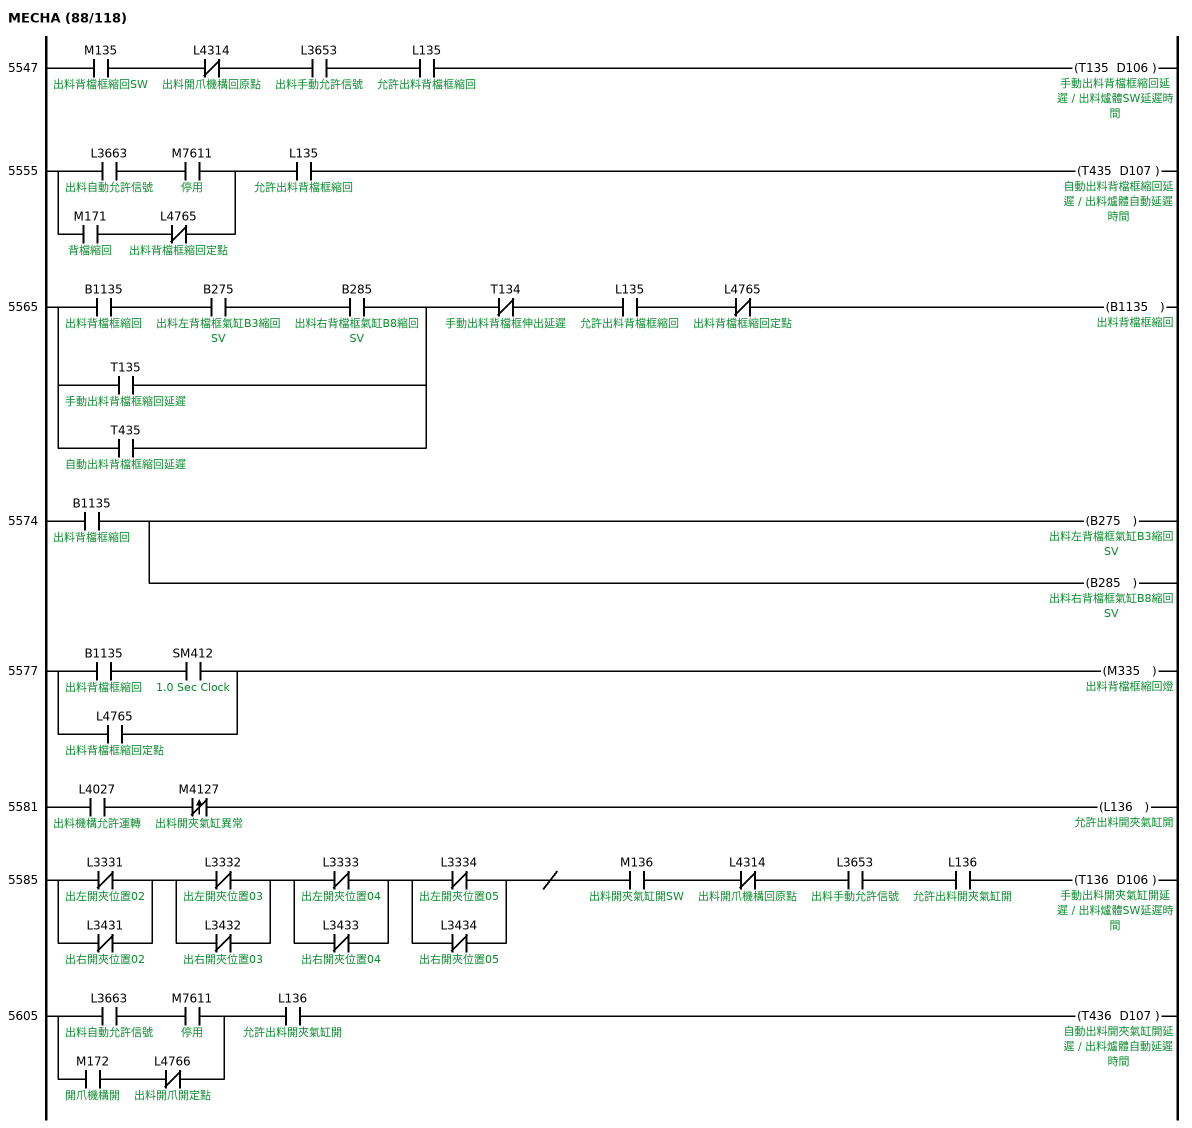
[picture p384: ladder of MECHA, rungs at steps 5547 to 5605]
5547  LD      M135  ; 出料背檔框縮回SW
      ANI     L4314  ; 出料開爪機構回原點
      AND     L3653  ; 出料手動允許信號
      AND     L135  ; 允許出料背檔框縮回
      OUT     T135 D106  ; 手動出料背檔框縮回延遲 / 出料爐體SW延遲時間
5555  LD      L3663  ; 出料自動允許信號
      AND     M7611  ; 停用
      LD      M171  ; 背檔縮回
      ANI     L4765  ; 出料背檔框縮回定點
      ORB
      AND     L135  ; 允許出料背檔框縮回
      OUT     T435 D107  ; 自動出料背檔框縮回延遲 / 出料爐體自動延遲時間
5565  LD      B1135  ; 出料背檔框縮回
      AND     B275  ; 出料左背檔框氣缸B3縮回SV
      AND     B285  ; 出料右背檔框氣缸B8縮回SV
      OR      T135  ; 手動出料背檔框縮回延遲
      OR      T435  ; 自動出料背檔框縮回延遲
      ANI     T134  ; 手動出料背檔框伸出延遲
      AND     L135  ; 允許出料背檔框縮回
      ANI     L4765  ; 出料背檔框縮回定點
      OUT     B1135  ; 出料背檔框縮回
5574  LD      B1135  ; 出料背檔框縮回
      OUT     B275  ; 出料左背檔框氣缸B3縮回SV
      OUT     B285  ; 出料右背檔框氣缸B8縮回SV
5577  LD      B1135  ; 出料背檔框縮回
      AND     SM412  ; 1.0 Sec Clock
      OR      L4765  ; 出料背檔框縮回定點
      OUT     M335  ; 出料背檔框縮回燈
5581  LD      L4027  ; 出料機構允許運轉
      ANDPI   M4127  ; 出料開夾氣缸異常
      OUT     L136  ; 允許出料開夾氣缸開
5585  LDI     L3331  ; 出左開夾位置02
      ORI     L3431  ; 出右開夾位置02
      LDI     L3332  ; 出左開夾位置03
      ORI     L3432  ; 出右開夾位置03
      ANB
      LDI     L3333  ; 出左開夾位置04
      ORI     L3433  ; 出右開夾位置04
      ANB
      LDI     L3334  ; 出左開夾位置05
      ORI     L3434  ; 出右開夾位置05
      ANB
      INV
      AND     M136  ; 出料開夾氣缸開SW
      ANI     L4314  ; 出料開爪機構回原點
      AND     L3653  ; 出料手動允許信號
      AND     L136  ; 允許出料開夾氣缸開
      OUT     T136 D106  ; 手動出料開夾氣缸開延遲 / 出料爐體SW延遲時間
5605  LD      L3663  ; 出料自動允許信號
      AND     M7611  ; 停用
      LD      M172  ; 開爪機構開
      ANI     L4766  ; 出料開爪開定點
      ORB
      AND     L136  ; 允許出料開夾氣缸開
      OUT     T436 D107  ; 自動出料開夾氣缸開延遲 / 出料爐體自動延遲時間
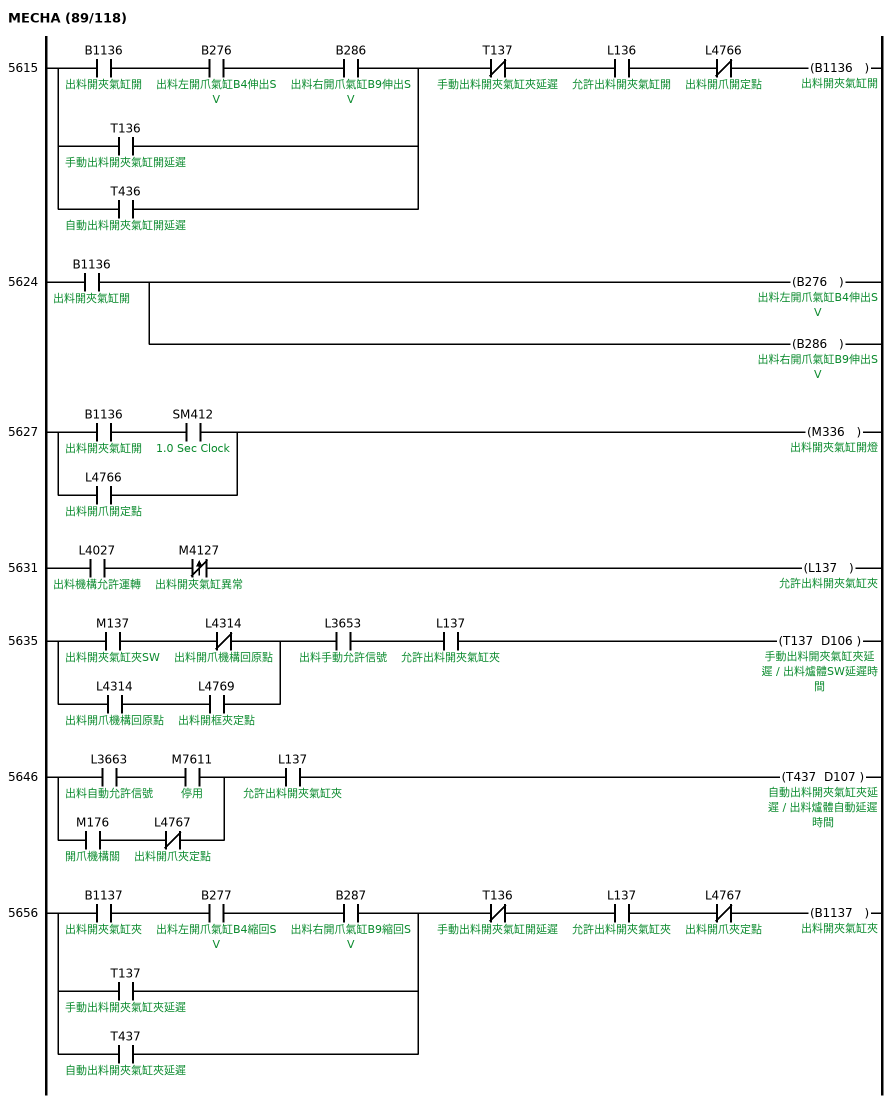
5615  LD      B1136  ; 出料開夾氣缸開
      AND     B276  ; 出料左開爪氣缸B4伸出SV
      AND     B286  ; 出料右開爪氣缸B9伸出SV
      OR      T136  ; 手動出料開夾氣缸開延遲
      OR      T436  ; 自動出料開夾氣缸開延遲
      ANI     T137  ; 手動出料開夾氣缸夾延遲
      AND     L136  ; 允許出料開夾氣缸開
      ANI     L4766  ; 出料開爪開定點
      OUT     B1136  ; 出料開夾氣缸開
5624  LD      B1136  ; 出料開夾氣缸開
      OUT     B276  ; 出料左開爪氣缸B4伸出SV
      OUT     B286  ; 出料右開爪氣缸B9伸出SV
5627  LD      B1136  ; 出料開夾氣缸開
      AND     SM412  ; 1.0 Sec Clock
      OR      L4766  ; 出料開爪開定點
      OUT     M336  ; 出料開夾氣缸開燈
5631  LD      L4027  ; 出料機構允許運轉
      ANDPI   M4127  ; 出料開夾氣缸異常
      OUT     L137  ; 允許出料開夾氣缸夾
5635  LD      M137  ; 出料開夾氣缸夾SW
      ANI     L4314  ; 出料開爪機構回原點
      LD      L4314  ; 出料開爪機構回原點
      AND     L4769  ; 出料開框夾定點
      ORB
      AND     L3653  ; 出料手動允許信號
      AND     L137  ; 允許出料開夾氣缸夾
      OUT     T137 D106  ; 手動出料開夾氣缸夾延遲 / 出料爐體SW延遲時間
5646  LD      L3663  ; 出料自動允許信號
      AND     M7611  ; 停用
      LD      M176  ; 開爪機構關
      ANI     L4767  ; 出料開爪夾定點
      ORB
      AND     L137  ; 允許出料開夾氣缸夾
      OUT     T437 D107  ; 自動出料開夾氣缸夾延遲 / 出料爐體自動延遲時間
5656  LD      B1137  ; 出料開夾氣缸夾
      AND     B277  ; 出料左開爪氣缸B4縮回SV
      AND     B287  ; 出料右開爪氣缸B9縮回SV
      OR      T137  ; 手動出料開夾氣缸夾延遲
      OR      T437  ; 自動出料開夾氣缸夾延遲
      ANI     T136  ; 手動出料開夾氣缸開延遲
      AND     L137  ; 允許出料開夾氣缸夾
      ANI     L4767  ; 出料開爪夾定點
      OUT     B1137  ; 出料開夾氣缸夾
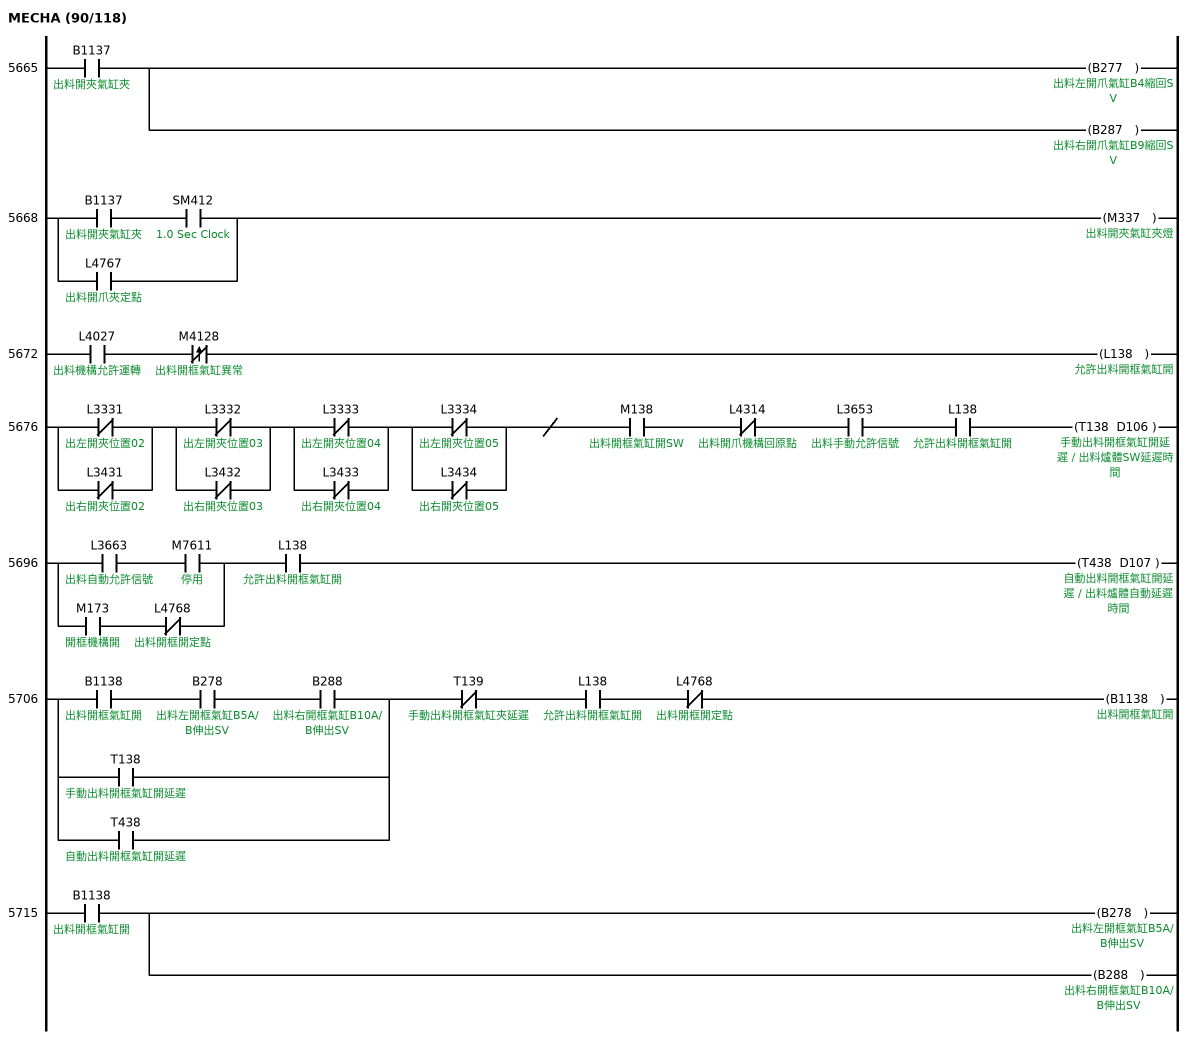
5665  LD      B1137  ; 出料開夾氣缸夾
      OUT     B277  ; 出料左開爪氣缸B4縮回SV
      OUT     B287  ; 出料右開爪氣缸B9縮回SV
5668  LD      B1137  ; 出料開夾氣缸夾
      AND     SM412  ; 1.0 Sec Clock
      OR      L4767  ; 出料開爪夾定點
      OUT     M337  ; 出料開夾氣缸夾燈
5672  LD      L4027  ; 出料機構允許運轉
      ANDPI   M4128  ; 出料開框氣缸異常
      OUT     L138  ; 允許出料開框氣缸開
5676  LDI     L3331  ; 出左開夾位置02
      ORI     L3431  ; 出右開夾位置02
      LDI     L3332  ; 出左開夾位置03
      ORI     L3432  ; 出右開夾位置03
      ANB
      LDI     L3333  ; 出左開夾位置04
      ORI     L3433  ; 出右開夾位置04
      ANB
      LDI     L3334  ; 出左開夾位置05
      ORI     L3434  ; 出右開夾位置05
      ANB
      INV
      AND     M138  ; 出料開框氣缸開SW
      ANI     L4314  ; 出料開爪機構回原點
      AND     L3653  ; 出料手動允許信號
      AND     L138  ; 允許出料開框氣缸開
      OUT     T138 D106  ; 手動出料開框氣缸開延遲 / 出料爐體SW延遲時間
5696  LD      L3663  ; 出料自動允許信號
      AND     M7611  ; 停用
      LD      M173  ; 開框機構開
      ANI     L4768  ; 出料開框開定點
      ORB
      AND     L138  ; 允許出料開框氣缸開
      OUT     T438 D107  ; 自動出料開框氣缸開延遲 / 出料爐體自動延遲時間
5706  LD      B1138  ; 出料開框氣缸開
      AND     B278  ; 出料左開框氣缸B5A/B伸出SV
      AND     B288  ; 出料右開框氣缸B10A/B伸出SV
      OR      T138  ; 手動出料開框氣缸開延遲
      OR      T438  ; 自動出料開框氣缸開延遲
      ANI     T139  ; 手動出料開框氣缸夾延遲
      AND     L138  ; 允許出料開框氣缸開
      ANI     L4768  ; 出料開框開定點
      OUT     B1138  ; 出料開框氣缸開
5715  LD      B1138  ; 出料開框氣缸開
      OUT     B278  ; 出料左開框氣缸B5A/B伸出SV
      OUT     B288  ; 出料右開框氣缸B10A/B伸出SV
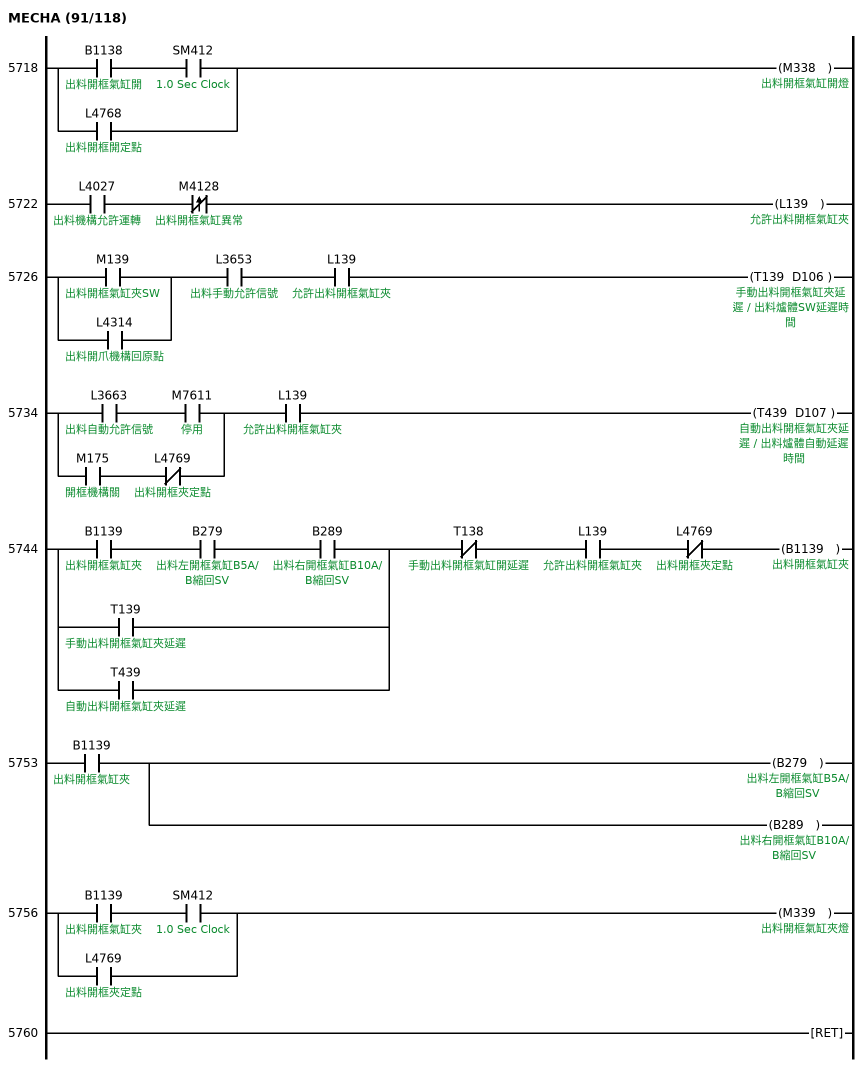
5718  LD      B1138  ; 出料開框氣缸開
      AND     SM412  ; 1.0 Sec Clock
      OR      L4768  ; 出料開框開定點
      OUT     M338  ; 出料開框氣缸開燈
5722  LD      L4027  ; 出料機構允許運轉
      ANDPI   M4128  ; 出料開框氣缸異常
      OUT     L139  ; 允許出料開框氣缸夾
5726  LD      M139  ; 出料開框氣缸夾SW
      OR      L4314  ; 出料開爪機構回原點
      AND     L3653  ; 出料手動允許信號
      AND     L139  ; 允許出料開框氣缸夾
      OUT     T139 D106  ; 手動出料開框氣缸夾延遲 / 出料爐體SW延遲時間
5734  LD      L3663  ; 出料自動允許信號
      AND     M7611  ; 停用
      LD      M175  ; 開框機構關
      ANI     L4769  ; 出料開框夾定點
      ORB
      AND     L139  ; 允許出料開框氣缸夾
      OUT     T439 D107  ; 自動出料開框氣缸夾延遲 / 出料爐體自動延遲時間
5744  LD      B1139  ; 出料開框氣缸夾
      AND     B279  ; 出料左開框氣缸B5A/B縮回SV
      AND     B289  ; 出料右開框氣缸B10A/B縮回SV
      OR      T139  ; 手動出料開框氣缸夾延遲
      OR      T439  ; 自動出料開框氣缸夾延遲
      ANI     T138  ; 手動出料開框氣缸開延遲
      AND     L139  ; 允許出料開框氣缸夾
      ANI     L4769  ; 出料開框夾定點
      OUT     B1139  ; 出料開框氣缸夾
5753  LD      B1139  ; 出料開框氣缸夾
      OUT     B279  ; 出料左開框氣缸B5A/B縮回SV
      OUT     B289  ; 出料右開框氣缸B10A/B縮回SV
5756  LD      B1139  ; 出料開框氣缸夾
      AND     SM412  ; 1.0 Sec Clock
      OR      L4769  ; 出料開框夾定點
      OUT     M339  ; 出料開框氣缸夾燈
5760  RET
      P1061
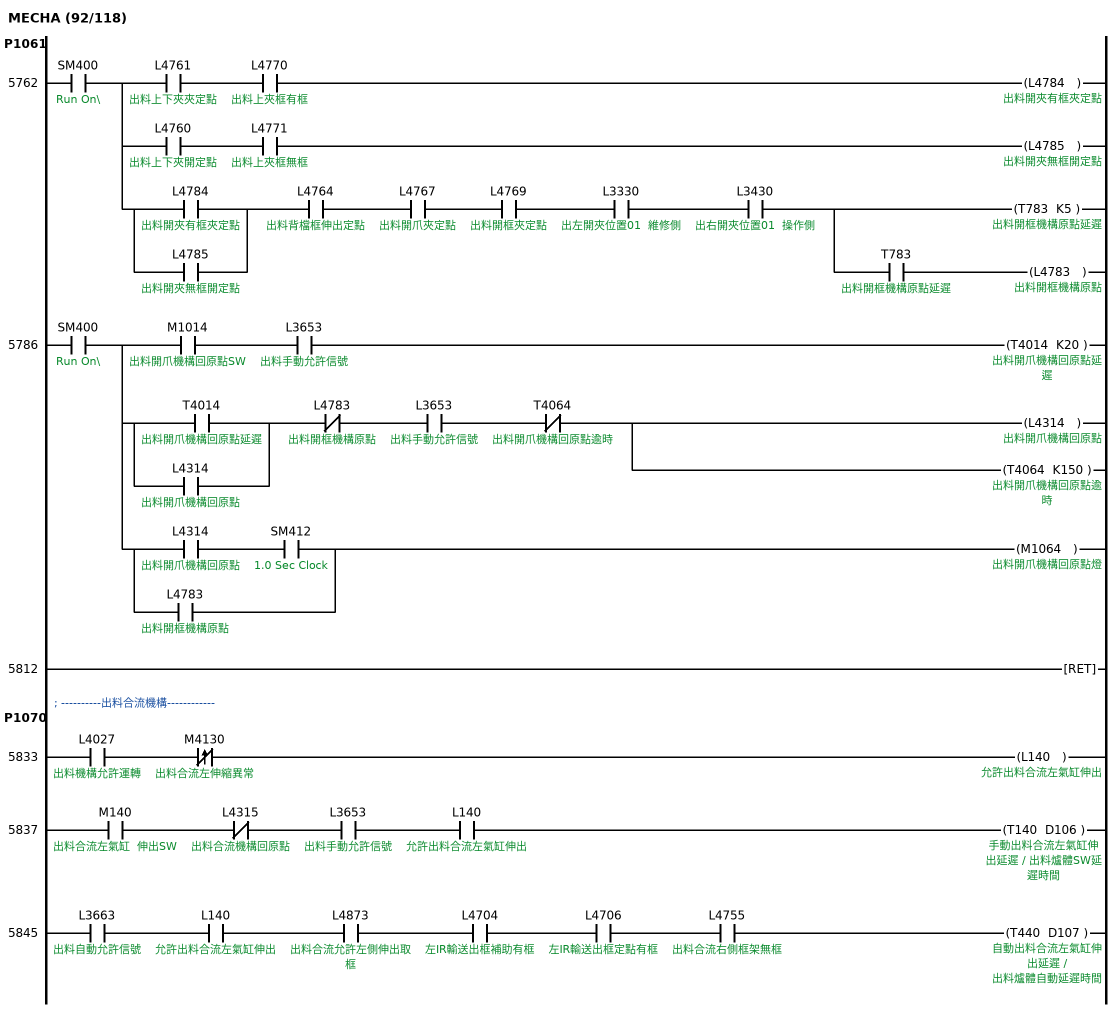
5762  LD      SM400  ; Run On\
      MPS
      AND     L4761  ; 出料上下夾夾定點
      AND     L4770  ; 出料上夾框有框
      OUT     L4784  ; 出料開夾有框夾定點
      MRD
      AND     L4760  ; 出料上下夾開定點
      AND     L4771  ; 出料上夾框無框
      OUT     L4785  ; 出料開夾無框開定點
      MPP
      LD      L4784  ; 出料開夾有框夾定點
      OR      L4785  ; 出料開夾無框開定點
      ANB
      AND     L4764  ; 出料背檔框伸出定點
      AND     L4767  ; 出料開爪夾定點
      AND     L4769  ; 出料開框夾定點
      AND     L3330  ; 出左開夾位置01  維修側
      AND     L3430  ; 出右開夾位置01  操作側
      OUT     T783 K5  ; 出料開框機構原點延遲
      AND     T783  ; 出料開框機構原點延遲
      OUT     L4783  ; 出料開框機構原點
5786  LD      SM400  ; Run On\
      MPS
      AND     M1014  ; 出料開爪機構回原點SW
      AND     L3653  ; 出料手動允許信號
      OUT     T4014 K20  ; 出料開爪機構回原點延遲
      MRD
      LD      T4014  ; 出料開爪機構回原點延遲
      OR      L4314  ; 出料開爪機構回原點
      ANB
      ANI     L4783  ; 出料開框機構原點
      AND     L3653  ; 出料手動允許信號
      ANI     T4064  ; 出料開爪機構回原點逾時
      OUT     L4314  ; 出料開爪機構回原點
      OUT     T4064 K150  ; 出料開爪機構回原點逾時
      MPP
      LD      L4314  ; 出料開爪機構回原點
      AND     SM412  ; 1.0 Sec Clock
      OR      L4783  ; 出料開框機構原點
      ANB
      OUT     M1064  ; 出料開爪機構回原點燈
5812  RET
; ----------出料合流機構------------
      P1070
5833  LD      L4027  ; 出料機構允許運轉
      ANDPI   M4130  ; 出料合流左伸縮異常
      OUT     L140  ; 允許出料合流左氣缸伸出
5837  LD      M140  ; 出料合流左氣缸  伸出SW
      ANI     L4315  ; 出料合流機構回原點
      AND     L3653  ; 出料手動允許信號
      AND     L140  ; 允許出料合流左氣缸伸出
      OUT     T140 D106  ; 手動出料合流左氣缸伸出延遲 / 出料爐體SW延遲時間
5845  LD      L3663  ; 出料自動允許信號
      AND     L140  ; 允許出料合流左氣缸伸出
      AND     L4873  ; 出料合流允許左側伸出取框
      AND     L4704  ; 左IR輸送出框補助有框
      AND     L4706  ; 左IR輸送出框定點有框
      AND     L4755  ; 出料合流右側框架無框
      OUT     T440 D107  ; 自動出料合流左氣缸伸出延遲 / 出料爐體自動延遲時間
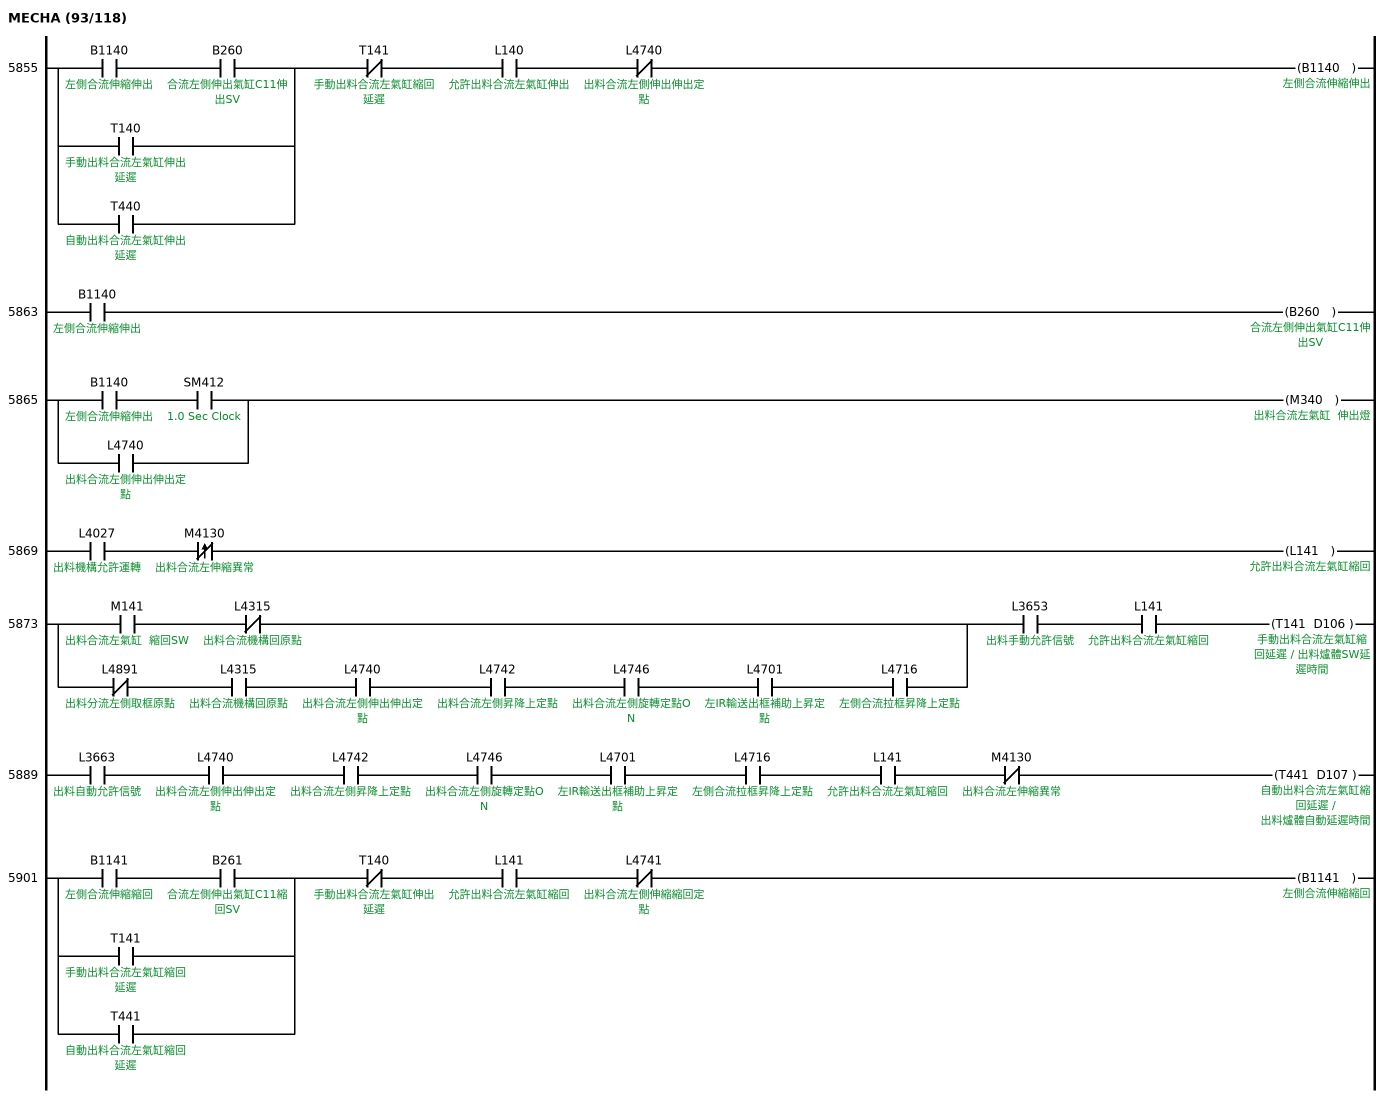
5855  LD      B1140  ; 左側合流伸縮伸出
      AND     B260  ; 合流左側伸出氣缸C11伸出SV
      OR      T140  ; 手動出料合流左氣缸伸出延遲
      OR      T440  ; 自動出料合流左氣缸伸出延遲
      ANI     T141  ; 手動出料合流左氣缸縮回延遲
      AND     L140  ; 允許出料合流左氣缸伸出
      ANI     L4740  ; 出料合流左側伸出伸出定點
      OUT     B1140  ; 左側合流伸縮伸出
5863  LD      B1140  ; 左側合流伸縮伸出
      OUT     B260  ; 合流左側伸出氣缸C11伸出SV
5865  LD      B1140  ; 左側合流伸縮伸出
      AND     SM412  ; 1.0 Sec Clock
      OR      L4740  ; 出料合流左側伸出伸出定點
      OUT     M340  ; 出料合流左氣缸  伸出燈
5869  LD      L4027  ; 出料機構允許運轉
      ANDPI   M4130  ; 出料合流左伸縮異常
      OUT     L141  ; 允許出料合流左氣缸縮回
5873  LD      M141  ; 出料合流左氣缸  縮回SW
      ANI     L4315  ; 出料合流機構回原點
      LDI     L4891  ; 出料分流左側取框原點
      AND     L4315  ; 出料合流機構回原點
      AND     L4740  ; 出料合流左側伸出伸出定點
      AND     L4742  ; 出料合流左側昇降上定點
      AND     L4746  ; 出料合流左側旋轉定點ON
      AND     L4701  ; 左IR輸送出框補助上昇定點
      AND     L4716  ; 左側合流拉框昇降上定點
      ORB
      AND     L3653  ; 出料手動允許信號
      AND     L141  ; 允許出料合流左氣缸縮回
      OUT     T141 D106  ; 手動出料合流左氣缸縮回延遲 / 出料爐體SW延遲時間
5889  LD      L3663  ; 出料自動允許信號
      AND     L4740  ; 出料合流左側伸出伸出定點
      AND     L4742  ; 出料合流左側昇降上定點
      AND     L4746  ; 出料合流左側旋轉定點ON
      AND     L4701  ; 左IR輸送出框補助上昇定點
      AND     L4716  ; 左側合流拉框昇降上定點
      AND     L141  ; 允許出料合流左氣缸縮回
      ANI     M4130  ; 出料合流左伸縮異常
      OUT     T441 D107  ; 自動出料合流左氣缸縮回延遲 / 出料爐體自動延遲時間
5901  LD      B1141  ; 左側合流伸縮縮回
      AND     B261  ; 合流左側伸出氣缸C11縮回SV
      OR      T141  ; 手動出料合流左氣缸縮回延遲
      OR      T441  ; 自動出料合流左氣缸縮回延遲
      ANI     T140  ; 手動出料合流左氣缸伸出延遲
      AND     L141  ; 允許出料合流左氣缸縮回
      ANI     L4741  ; 出料合流左側伸縮縮回定點
      OUT     B1141  ; 左側合流伸縮縮回
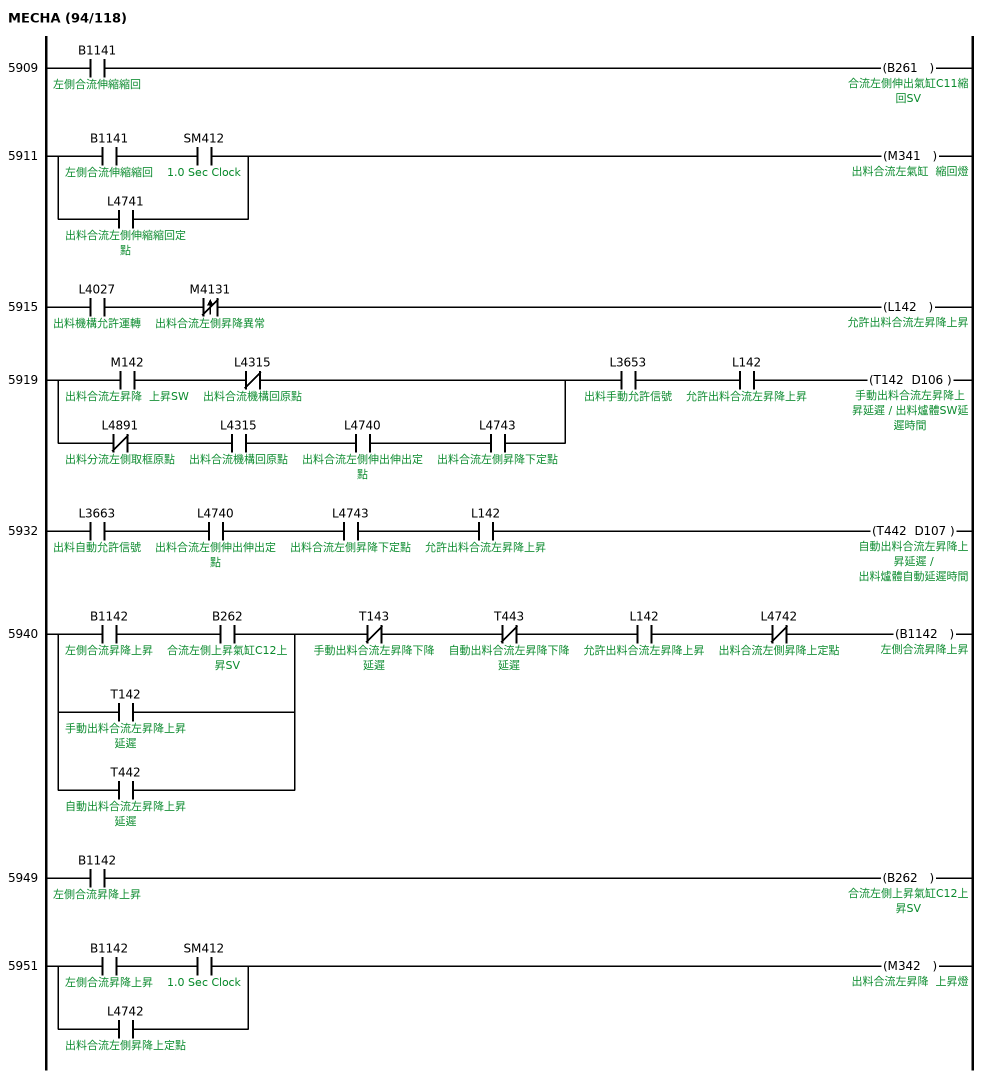
5909  LD      B1141  ; 左側合流伸縮縮回
      OUT     B261  ; 合流左側伸出氣缸C11縮回SV
5911  LD      B1141  ; 左側合流伸縮縮回
      AND     SM412  ; 1.0 Sec Clock
      OR      L4741  ; 出料合流左側伸縮縮回定點
      OUT     M341  ; 出料合流左氣缸  縮回燈
5915  LD      L4027  ; 出料機構允許運轉
      ANDPI   M4131  ; 出料合流左側昇降異常
      OUT     L142  ; 允許出料合流左昇降上昇
5919  LD      M142  ; 出料合流左昇降  上昇SW
      ANI     L4315  ; 出料合流機構回原點
      LDI     L4891  ; 出料分流左側取框原點
      AND     L4315  ; 出料合流機構回原點
      AND     L4740  ; 出料合流左側伸出伸出定點
      AND     L4743  ; 出料合流左側昇降下定點
      ORB
      AND     L3653  ; 出料手動允許信號
      AND     L142  ; 允許出料合流左昇降上昇
      OUT     T142 D106  ; 手動出料合流左昇降上昇延遲 / 出料爐體SW延遲時間
5932  LD      L3663  ; 出料自動允許信號
      AND     L4740  ; 出料合流左側伸出伸出定點
      AND     L4743  ; 出料合流左側昇降下定點
      AND     L142  ; 允許出料合流左昇降上昇
      OUT     T442 D107  ; 自動出料合流左昇降上昇延遲 / 出料爐體自動延遲時間
5940  LD      B1142  ; 左側合流昇降上昇
      AND     B262  ; 合流左側上昇氣缸C12上昇SV
      OR      T142  ; 手動出料合流左昇降上昇延遲
      OR      T442  ; 自動出料合流左昇降上昇延遲
      ANI     T143  ; 手動出料合流左昇降下降延遲
      ANI     T443  ; 自動出料合流左昇降下降延遲
      AND     L142  ; 允許出料合流左昇降上昇
      ANI     L4742  ; 出料合流左側昇降上定點
      OUT     B1142  ; 左側合流昇降上昇
5949  LD      B1142  ; 左側合流昇降上昇
      OUT     B262  ; 合流左側上昇氣缸C12上昇SV
5951  LD      B1142  ; 左側合流昇降上昇
      AND     SM412  ; 1.0 Sec Clock
      OR      L4742  ; 出料合流左側昇降上定點
      OUT     M342  ; 出料合流左昇降  上昇燈
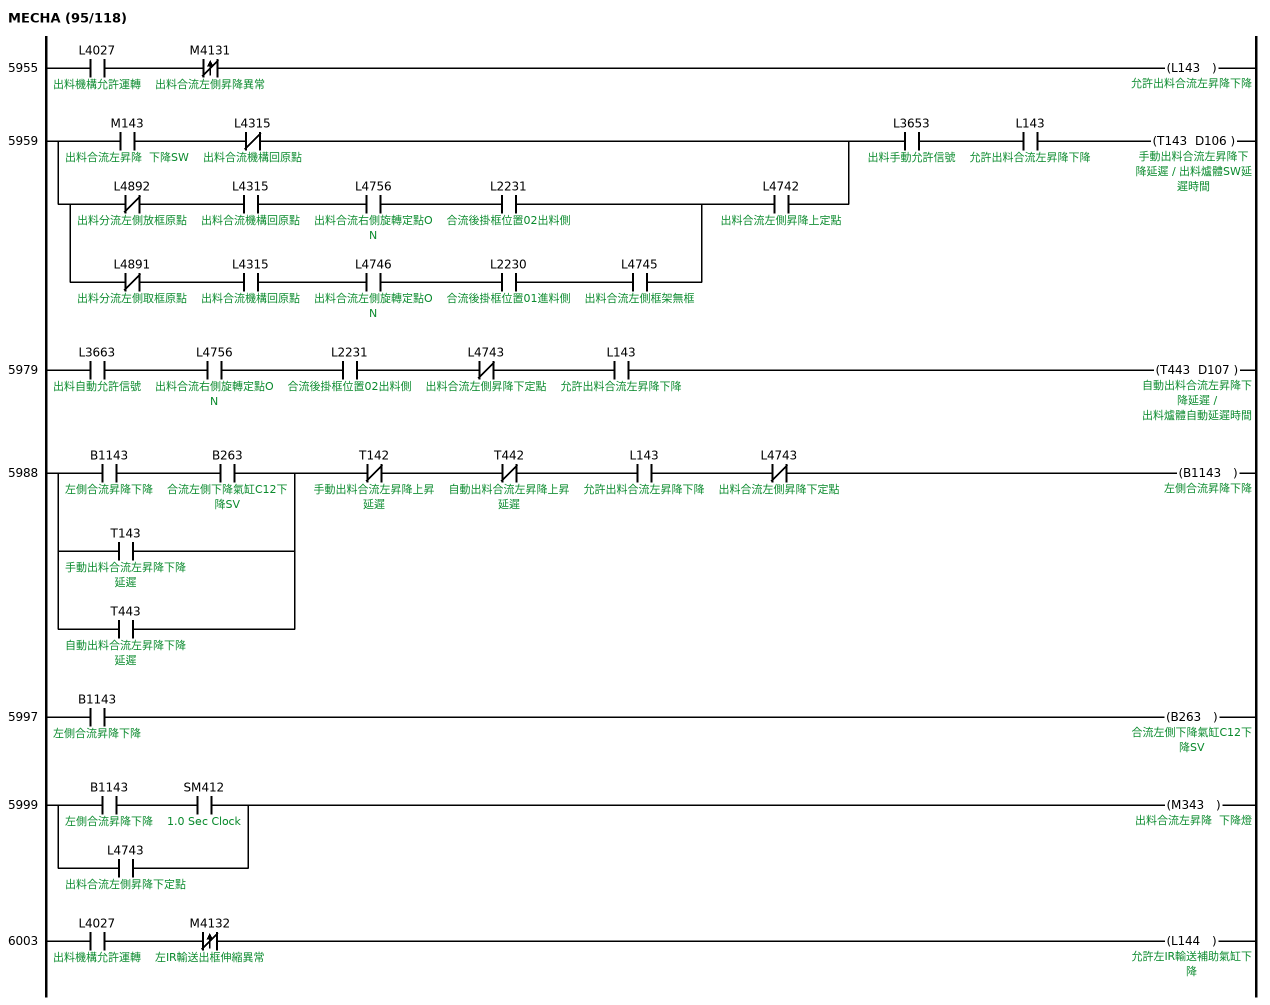
5955  LD      L4027  ; 出料機構允許運轉
      ANDPI   M4131  ; 出料合流左側昇降異常
      OUT     L143  ; 允許出料合流左昇降下降
5959  LD      M143  ; 出料合流左昇降  下降SW
      ANI     L4315  ; 出料合流機構回原點
      LDI     L4892  ; 出料分流左側放框原點
      AND     L4315  ; 出料合流機構回原點
      AND     L4756  ; 出料合流右側旋轉定點ON
      AND     L2231  ; 合流後掛框位置02出料側
      LDI     L4891  ; 出料分流左側取框原點
      AND     L4315  ; 出料合流機構回原點
      AND     L4746  ; 出料合流左側旋轉定點ON
      AND     L2230  ; 合流後掛框位置01進料側
      AND     L4745  ; 出料合流左側框架無框
      ORB
      AND     L4742  ; 出料合流左側昇降上定點
      ORB
      AND     L3653  ; 出料手動允許信號
      AND     L143  ; 允許出料合流左昇降下降
      OUT     T143 D106  ; 手動出料合流左昇降下降延遲 / 出料爐體SW延遲時間
5979  LD      L3663  ; 出料自動允許信號
      AND     L4756  ; 出料合流右側旋轉定點ON
      AND     L2231  ; 合流後掛框位置02出料側
      ANI     L4743  ; 出料合流左側昇降下定點
      AND     L143  ; 允許出料合流左昇降下降
      OUT     T443 D107  ; 自動出料合流左昇降下降延遲 / 出料爐體自動延遲時間
5988  LD      B1143  ; 左側合流昇降下降
      AND     B263  ; 合流左側下降氣缸C12下降SV
      OR      T143  ; 手動出料合流左昇降下降延遲
      OR      T443  ; 自動出料合流左昇降下降延遲
      ANI     T142  ; 手動出料合流左昇降上昇延遲
      ANI     T442  ; 自動出料合流左昇降上昇延遲
      AND     L143  ; 允許出料合流左昇降下降
      ANI     L4743  ; 出料合流左側昇降下定點
      OUT     B1143  ; 左側合流昇降下降
5997  LD      B1143  ; 左側合流昇降下降
      OUT     B263  ; 合流左側下降氣缸C12下降SV
5999  LD      B1143  ; 左側合流昇降下降
      AND     SM412  ; 1.0 Sec Clock
      OR      L4743  ; 出料合流左側昇降下定點
      OUT     M343  ; 出料合流左昇降  下降燈
6003  LD      L4027  ; 出料機構允許運轉
      ANDPI   M4132  ; 左IR輸送出框伸縮異常
      OUT     L144  ; 允許左IR輸送補助氣缸下降
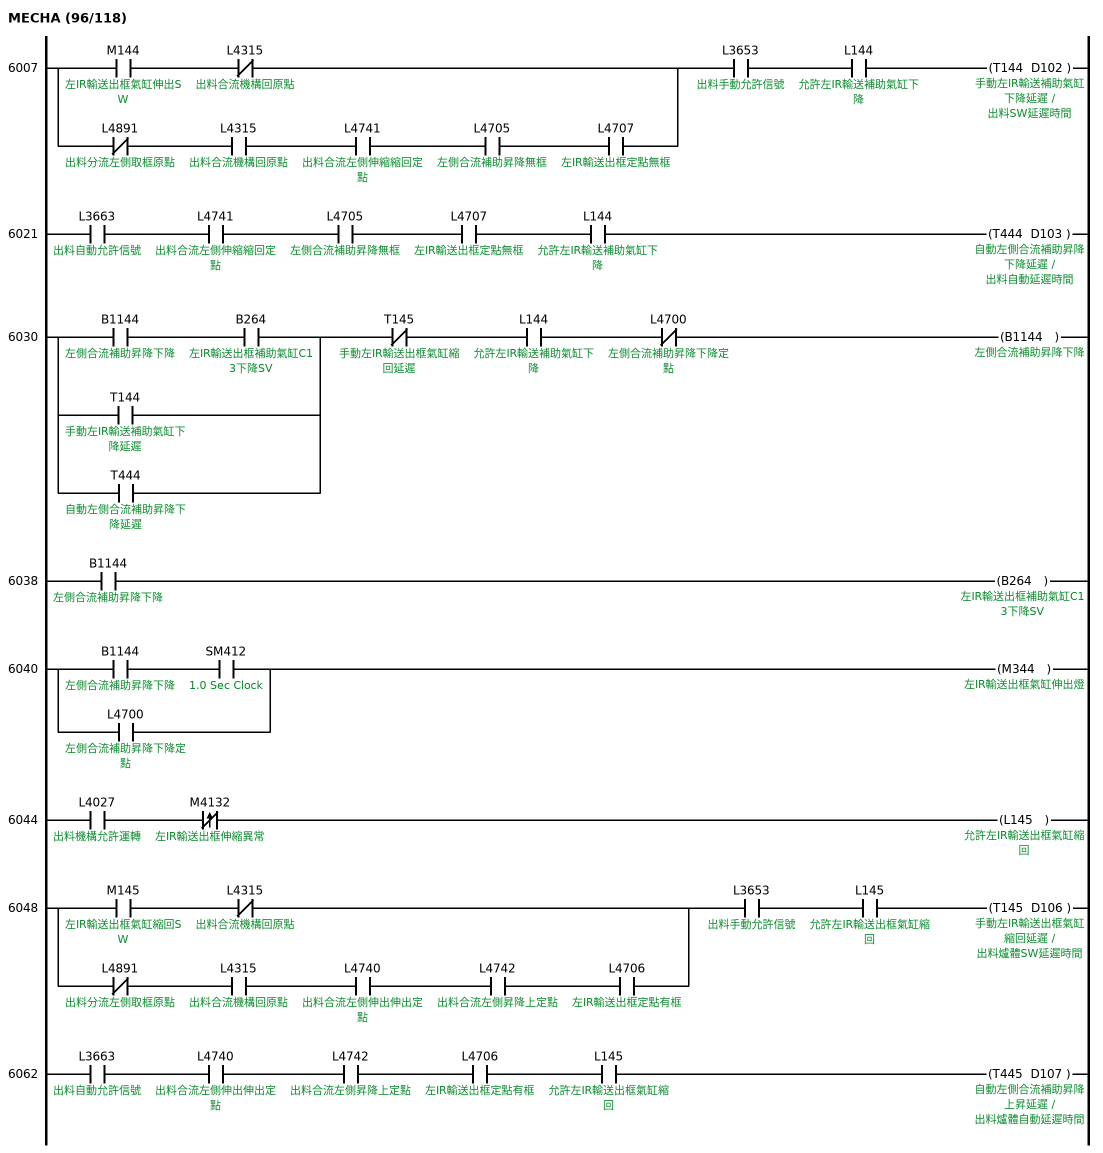
6007  LD      M144  ; 左IR輸送出框氣缸伸出SW
      ANI     L4315  ; 出料合流機構回原點
      LDI     L4891  ; 出料分流左側取框原點
      AND     L4315  ; 出料合流機構回原點
      AND     L4741  ; 出料合流左側伸縮縮回定點
      AND     L4705  ; 左側合流補助昇降無框
      AND     L4707  ; 左IR輸送出框定點無框
      ORB
      AND     L3653  ; 出料手動允許信號
      AND     L144  ; 允許左IR輸送補助氣缸下降
      OUT     T144 D102  ; 手動左IR輸送補助氣缸下降延遲 / 出料SW延遲時間
6021  LD      L3663  ; 出料自動允許信號
      AND     L4741  ; 出料合流左側伸縮縮回定點
      AND     L4705  ; 左側合流補助昇降無框
      AND     L4707  ; 左IR輸送出框定點無框
      AND     L144  ; 允許左IR輸送補助氣缸下降
      OUT     T444 D103  ; 自動左側合流補助昇降下降延遲 / 出料自動延遲時間
6030  LD      B1144  ; 左側合流補助昇降下降
      AND     B264  ; 左IR輸送出框補助氣缸C13下降SV
      OR      T144  ; 手動左IR輸送補助氣缸下降延遲
      OR      T444  ; 自動左側合流補助昇降下降延遲
      ANI     T145  ; 手動左IR輸送出框氣缸縮回延遲
      AND     L144  ; 允許左IR輸送補助氣缸下降
      ANI     L4700  ; 左側合流補助昇降下降定點
      OUT     B1144  ; 左側合流補助昇降下降
6038  LD      B1144  ; 左側合流補助昇降下降
      OUT     B264  ; 左IR輸送出框補助氣缸C13下降SV
6040  LD      B1144  ; 左側合流補助昇降下降
      AND     SM412  ; 1.0 Sec Clock
      OR      L4700  ; 左側合流補助昇降下降定點
      OUT     M344  ; 左IR輸送出框氣缸伸出燈
6044  LD      L4027  ; 出料機構允許運轉
      ANDPI   M4132  ; 左IR輸送出框伸縮異常
      OUT     L145  ; 允許左IR輸送出框氣缸縮回
6048  LD      M145  ; 左IR輸送出框氣缸縮回SW
      ANI     L4315  ; 出料合流機構回原點
      LDI     L4891  ; 出料分流左側取框原點
      AND     L4315  ; 出料合流機構回原點
      AND     L4740  ; 出料合流左側伸出伸出定點
      AND     L4742  ; 出料合流左側昇降上定點
      AND     L4706  ; 左IR輸送出框定點有框
      ORB
      AND     L3653  ; 出料手動允許信號
      AND     L145  ; 允許左IR輸送出框氣缸縮回
      OUT     T145 D106  ; 手動左IR輸送出框氣缸縮回延遲 / 出料爐體SW延遲時間
6062  LD      L3663  ; 出料自動允許信號
      AND     L4740  ; 出料合流左側伸出伸出定點
      AND     L4742  ; 出料合流左側昇降上定點
      AND     L4706  ; 左IR輸送出框定點有框
      AND     L145  ; 允許左IR輸送出框氣缸縮回
      OUT     T445 D107  ; 自動左側合流補助昇降上昇延遲 / 出料爐體自動延遲時間
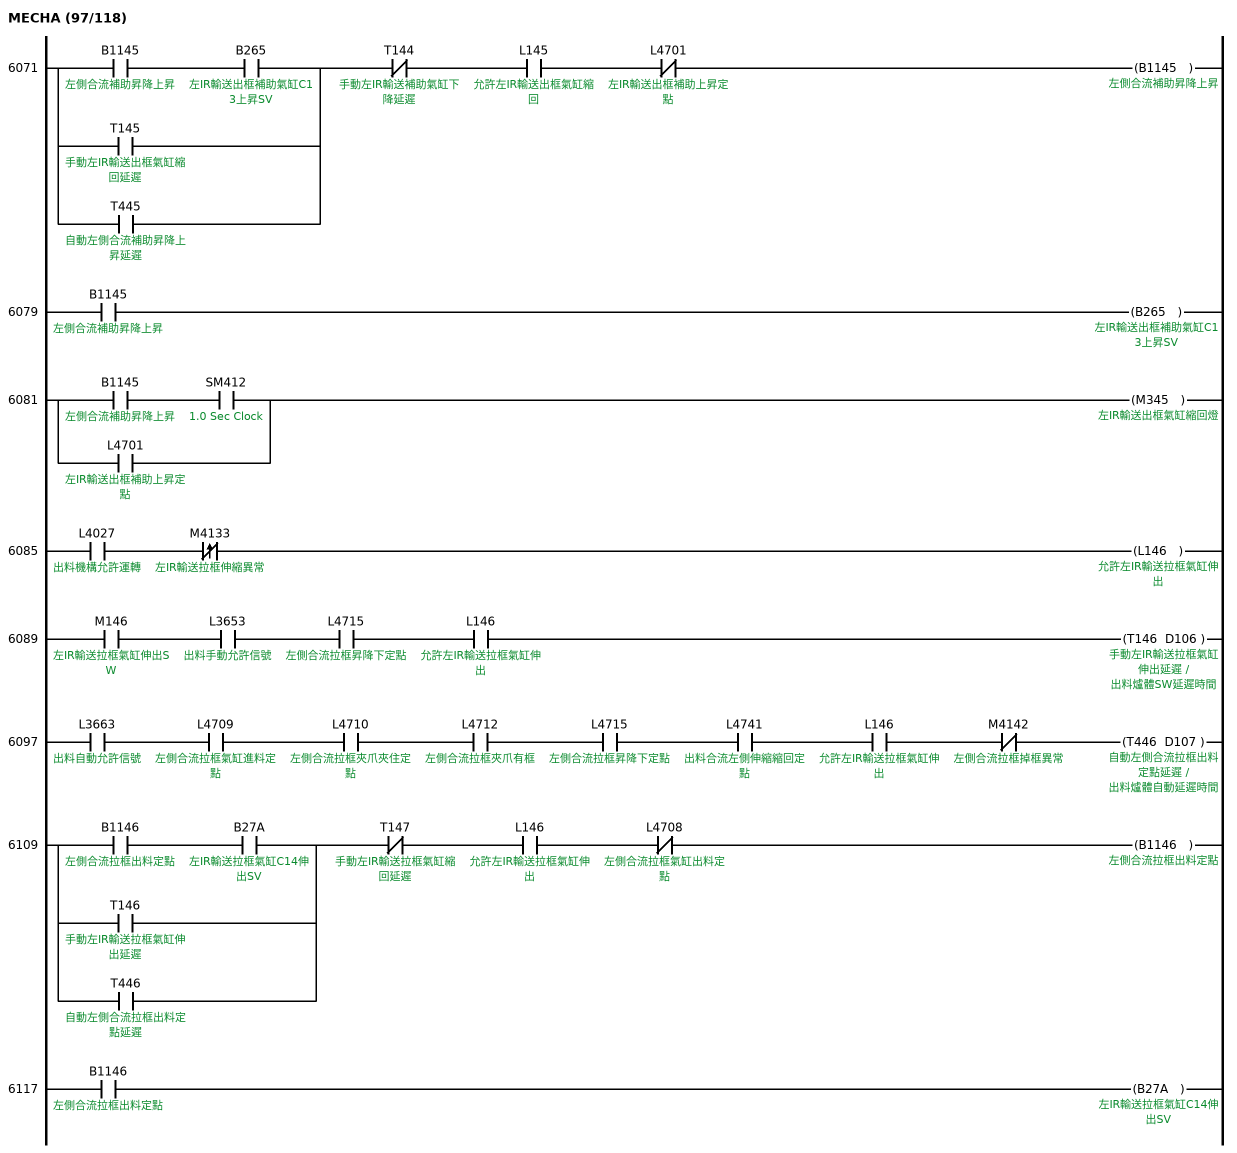
6071  LD      B1145  ; 左側合流補助昇降上昇
      AND     B265  ; 左IR輸送出框補助氣缸C13上昇SV
      OR      T145  ; 手動左IR輸送出框氣缸縮回延遲
      OR      T445  ; 自動左側合流補助昇降上昇延遲
      ANI     T144  ; 手動左IR輸送補助氣缸下降延遲
      AND     L145  ; 允許左IR輸送出框氣缸縮回
      ANI     L4701  ; 左IR輸送出框補助上昇定點
      OUT     B1145  ; 左側合流補助昇降上昇
6079  LD      B1145  ; 左側合流補助昇降上昇
      OUT     B265  ; 左IR輸送出框補助氣缸C13上昇SV
6081  LD      B1145  ; 左側合流補助昇降上昇
      AND     SM412  ; 1.0 Sec Clock
      OR      L4701  ; 左IR輸送出框補助上昇定點
      OUT     M345  ; 左IR輸送出框氣缸縮回燈
6085  LD      L4027  ; 出料機構允許運轉
      ANDPI   M4133  ; 左IR輸送拉框伸縮異常
      OUT     L146  ; 允許左IR輸送拉框氣缸伸出
6089  LD      M146  ; 左IR輸送拉框氣缸伸出SW
      AND     L3653  ; 出料手動允許信號
      AND     L4715  ; 左側合流拉框昇降下定點
      AND     L146  ; 允許左IR輸送拉框氣缸伸出
      OUT     T146 D106  ; 手動左IR輸送拉框氣缸伸出延遲 / 出料爐體SW延遲時間
6097  LD      L3663  ; 出料自動允許信號
      AND     L4709  ; 左側合流拉框氣缸進料定點
      AND     L4710  ; 左側合流拉框夾爪夾住定點
      AND     L4712  ; 左側合流拉框夾爪有框
      AND     L4715  ; 左側合流拉框昇降下定點
      AND     L4741  ; 出料合流左側伸縮縮回定點
      AND     L146  ; 允許左IR輸送拉框氣缸伸出
      ANI     M4142  ; 左側合流拉框掉框異常
      OUT     T446 D107  ; 自動左側合流拉框出料定點延遲 / 出料爐體自動延遲時間
6109  LD      B1146  ; 左側合流拉框出料定點
      AND     B27A  ; 左IR輸送拉框氣缸C14伸出SV
      OR      T146  ; 手動左IR輸送拉框氣缸伸出延遲
      OR      T446  ; 自動左側合流拉框出料定點延遲
      ANI     T147  ; 手動左IR輸送拉框氣缸縮回延遲
      AND     L146  ; 允許左IR輸送拉框氣缸伸出
      ANI     L4708  ; 左側合流拉框氣缸出料定點
      OUT     B1146  ; 左側合流拉框出料定點
6117  LD      B1146  ; 左側合流拉框出料定點
      OUT     B27A  ; 左IR輸送拉框氣缸C14伸出SV
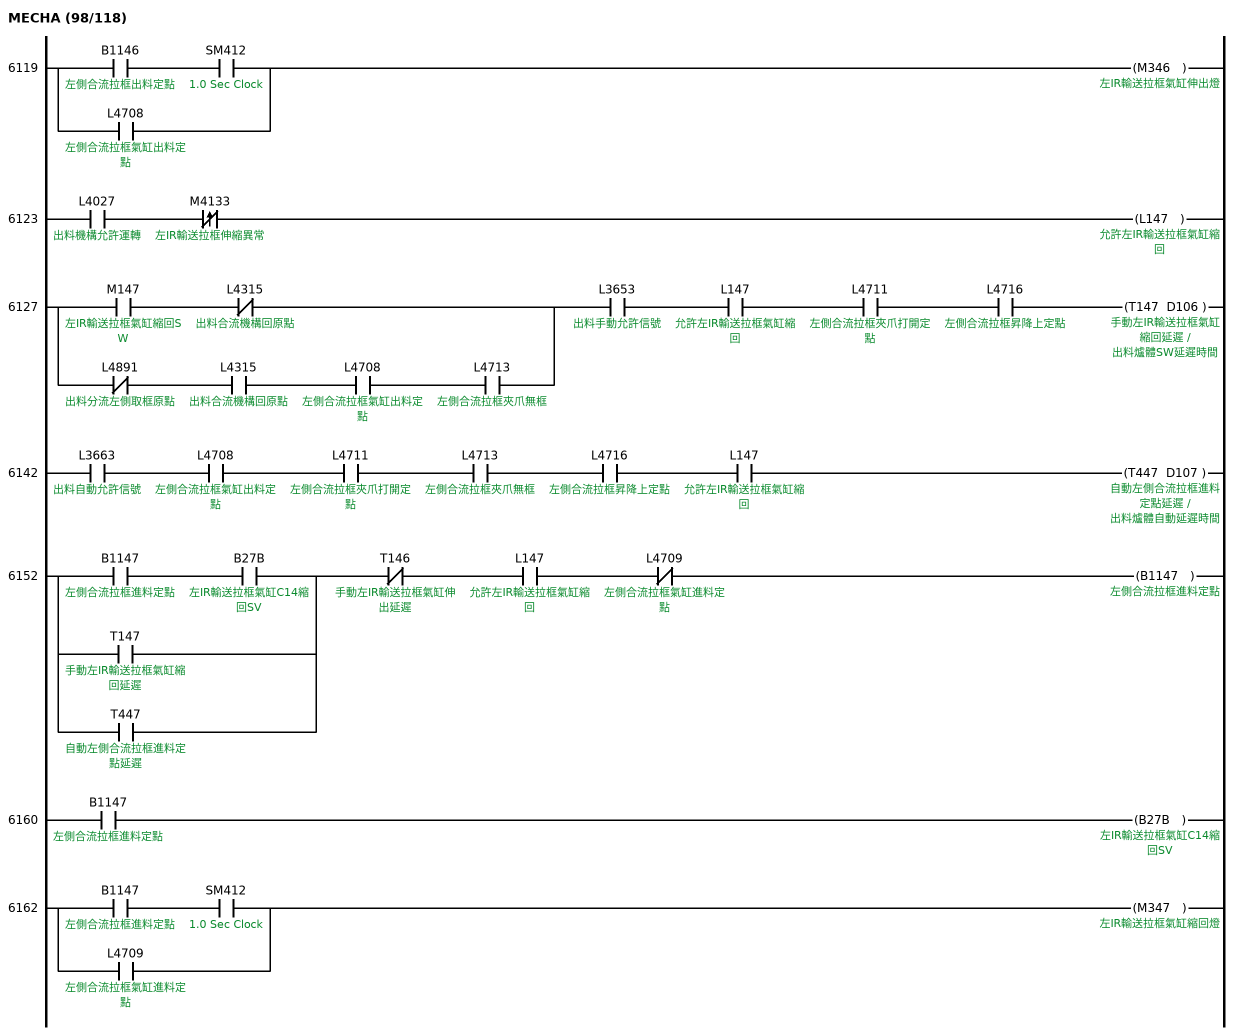
6119  LD      B1146  ; 左側合流拉框出料定點
      AND     SM412  ; 1.0 Sec Clock
      OR      L4708  ; 左側合流拉框氣缸出料定點
      OUT     M346  ; 左IR輸送拉框氣缸伸出燈
6123  LD      L4027  ; 出料機構允許運轉
      ANDPI   M4133  ; 左IR輸送拉框伸縮異常
      OUT     L147  ; 允許左IR輸送拉框氣缸縮回
6127  LD      M147  ; 左IR輸送拉框氣缸縮回SW
      ANI     L4315  ; 出料合流機構回原點
      LDI     L4891  ; 出料分流左側取框原點
      AND     L4315  ; 出料合流機構回原點
      AND     L4708  ; 左側合流拉框氣缸出料定點
      AND     L4713  ; 左側合流拉框夾爪無框
      ORB
      AND     L3653  ; 出料手動允許信號
      AND     L147  ; 允許左IR輸送拉框氣缸縮回
      AND     L4711  ; 左側合流拉框夾爪打開定點
      AND     L4716  ; 左側合流拉框昇降上定點
      OUT     T147 D106  ; 手動左IR輸送拉框氣缸縮回延遲 / 出料爐體SW延遲時間
6142  LD      L3663  ; 出料自動允許信號
      AND     L4708  ; 左側合流拉框氣缸出料定點
      AND     L4711  ; 左側合流拉框夾爪打開定點
      AND     L4713  ; 左側合流拉框夾爪無框
      AND     L4716  ; 左側合流拉框昇降上定點
      AND     L147  ; 允許左IR輸送拉框氣缸縮回
      OUT     T447 D107  ; 自動左側合流拉框進料定點延遲 / 出料爐體自動延遲時間
6152  LD      B1147  ; 左側合流拉框進料定點
      AND     B27B  ; 左IR輸送拉框氣缸C14縮回SV
      OR      T147  ; 手動左IR輸送拉框氣缸縮回延遲
      OR      T447  ; 自動左側合流拉框進料定點延遲
      ANI     T146  ; 手動左IR輸送拉框氣缸伸出延遲
      AND     L147  ; 允許左IR輸送拉框氣缸縮回
      ANI     L4709  ; 左側合流拉框氣缸進料定點
      OUT     B1147  ; 左側合流拉框進料定點
6160  LD      B1147  ; 左側合流拉框進料定點
      OUT     B27B  ; 左IR輸送拉框氣缸C14縮回SV
6162  LD      B1147  ; 左側合流拉框進料定點
      AND     SM412  ; 1.0 Sec Clock
      OR      L4709  ; 左側合流拉框氣缸進料定點
      OUT     M347  ; 左IR輸送拉框氣缸縮回燈
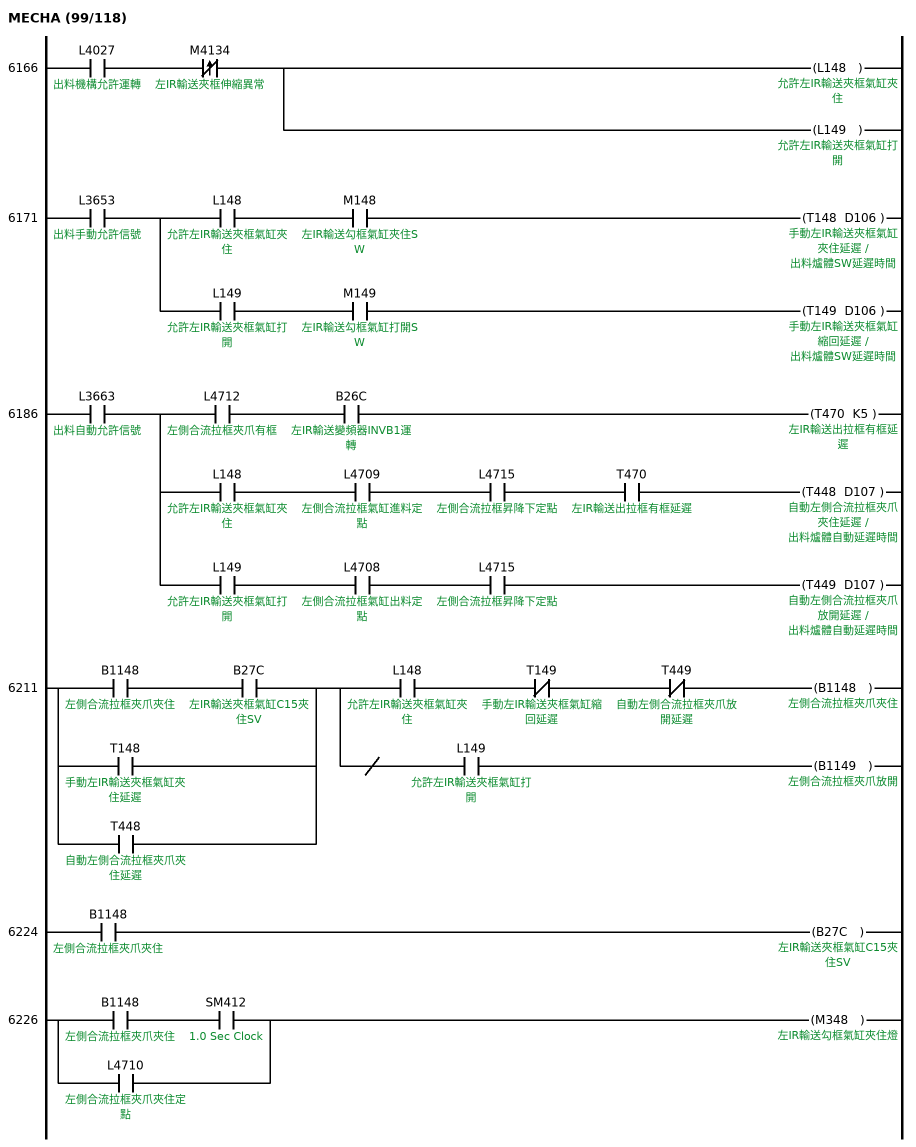
6166  LD      L4027  ; 出料機構允許運轉
      ANDPI   M4134  ; 左IR輸送夾框伸縮異常
      OUT     L148  ; 允許左IR輸送夾框氣缸夾住
      OUT     L149  ; 允許左IR輸送夾框氣缸打開
6171  LD      L3653  ; 出料手動允許信號
      MPS
      AND     L148  ; 允許左IR輸送夾框氣缸夾住
      AND     M148  ; 左IR輸送勾框氣缸夾住SW
      OUT     T148 D106  ; 手動左IR輸送夾框氣缸夾住延遲 / 出料爐體SW延遲時間
      MPP
      AND     L149  ; 允許左IR輸送夾框氣缸打開
      AND     M149  ; 左IR輸送勾框氣缸打開SW
      OUT     T149 D106  ; 手動左IR輸送夾框氣缸縮回延遲 / 出料爐體SW延遲時間
6186  LD      L3663  ; 出料自動允許信號
      MPS
      AND     L4712  ; 左側合流拉框夾爪有框
      AND     B26C  ; 左IR輸送變頻器INVB1運轉
      OUT     T470 K5  ; 左IR輸送出拉框有框延遲
      MRD
      AND     L148  ; 允許左IR輸送夾框氣缸夾住
      AND     L4709  ; 左側合流拉框氣缸進料定點
      AND     L4715  ; 左側合流拉框昇降下定點
      AND     T470  ; 左IR輸送出拉框有框延遲
      OUT     T448 D107  ; 自動左側合流拉框夾爪夾住延遲 / 出料爐體自動延遲時間
      MPP
      AND     L149  ; 允許左IR輸送夾框氣缸打開
      AND     L4708  ; 左側合流拉框氣缸出料定點
      AND     L4715  ; 左側合流拉框昇降下定點
      OUT     T449 D107  ; 自動左側合流拉框夾爪放開延遲 / 出料爐體自動延遲時間
6211  LD      B1148  ; 左側合流拉框夾爪夾住
      AND     B27C  ; 左IR輸送夾框氣缸C15夾住SV
      OR      T148  ; 手動左IR輸送夾框氣缸夾住延遲
      OR      T448  ; 自動左側合流拉框夾爪夾住延遲
      MPS
      AND     L148  ; 允許左IR輸送夾框氣缸夾住
      ANI     T149  ; 手動左IR輸送夾框氣缸縮回延遲
      ANI     T449  ; 自動左側合流拉框夾爪放開延遲
      OUT     B1148  ; 左側合流拉框夾爪夾住
      MPP
      INV
      AND     L149  ; 允許左IR輸送夾框氣缸打開
      OUT     B1149  ; 左側合流拉框夾爪放開
6224  LD      B1148  ; 左側合流拉框夾爪夾住
      OUT     B27C  ; 左IR輸送夾框氣缸C15夾住SV
6226  LD      B1148  ; 左側合流拉框夾爪夾住
      AND     SM412  ; 1.0 Sec Clock
      OR      L4710  ; 左側合流拉框夾爪夾住定點
      OUT     M348  ; 左IR輸送勾框氣缸夾住燈
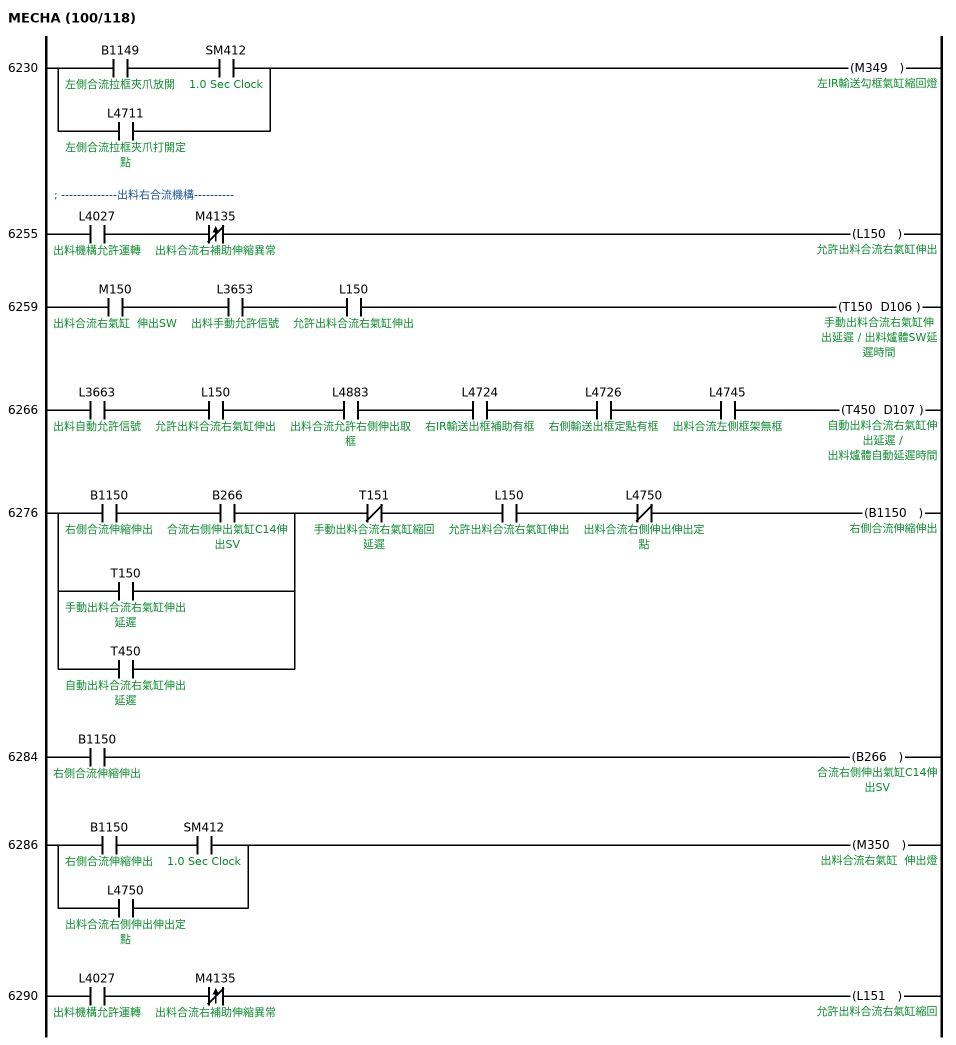
6230  LD      B1149  ; 左側合流拉框夾爪放開
      AND     SM412  ; 1.0 Sec Clock
      OR      L4711  ; 左側合流拉框夾爪打開定點
      OUT     M349  ; 左IR輸送勾框氣缸縮回燈
; --------------出料右合流機構----------
6255  LD      L4027  ; 出料機構允許運轉
      ANDPI   M4135  ; 出料合流右補助伸縮異常
      OUT     L150  ; 允許出料合流右氣缸伸出
6259  LD      M150  ; 出料合流右氣缸  伸出SW
      AND     L3653  ; 出料手動允許信號
      AND     L150  ; 允許出料合流右氣缸伸出
      OUT     T150 D106  ; 手動出料合流右氣缸伸出延遲 / 出料爐體SW延遲時間
6266  LD      L3663  ; 出料自動允許信號
      AND     L150  ; 允許出料合流右氣缸伸出
      AND     L4883  ; 出料合流允許右側伸出取框
      AND     L4724  ; 右IR輸送出框補助有框
      AND     L4726  ; 右側輸送出框定點有框
      AND     L4745  ; 出料合流左側框架無框
      OUT     T450 D107  ; 自動出料合流右氣缸伸出延遲 / 出料爐體自動延遲時間
6276  LD      B1150  ; 右側合流伸縮伸出
      AND     B266  ; 合流右側伸出氣缸C14伸出SV
      OR      T150  ; 手動出料合流右氣缸伸出延遲
      OR      T450  ; 自動出料合流右氣缸伸出延遲
      ANI     T151  ; 手動出料合流右氣缸縮回延遲
      AND     L150  ; 允許出料合流右氣缸伸出
      ANI     L4750  ; 出料合流右側伸出伸出定點
      OUT     B1150  ; 右側合流伸縮伸出
6284  LD      B1150  ; 右側合流伸縮伸出
      OUT     B266  ; 合流右側伸出氣缸C14伸出SV
6286  LD      B1150  ; 右側合流伸縮伸出
      AND     SM412  ; 1.0 Sec Clock
      OR      L4750  ; 出料合流右側伸出伸出定點
      OUT     M350  ; 出料合流右氣缸  伸出燈
6290  LD      L4027  ; 出料機構允許運轉
      ANDPI   M4135  ; 出料合流右補助伸縮異常
      OUT     L151  ; 允許出料合流右氣缸縮回
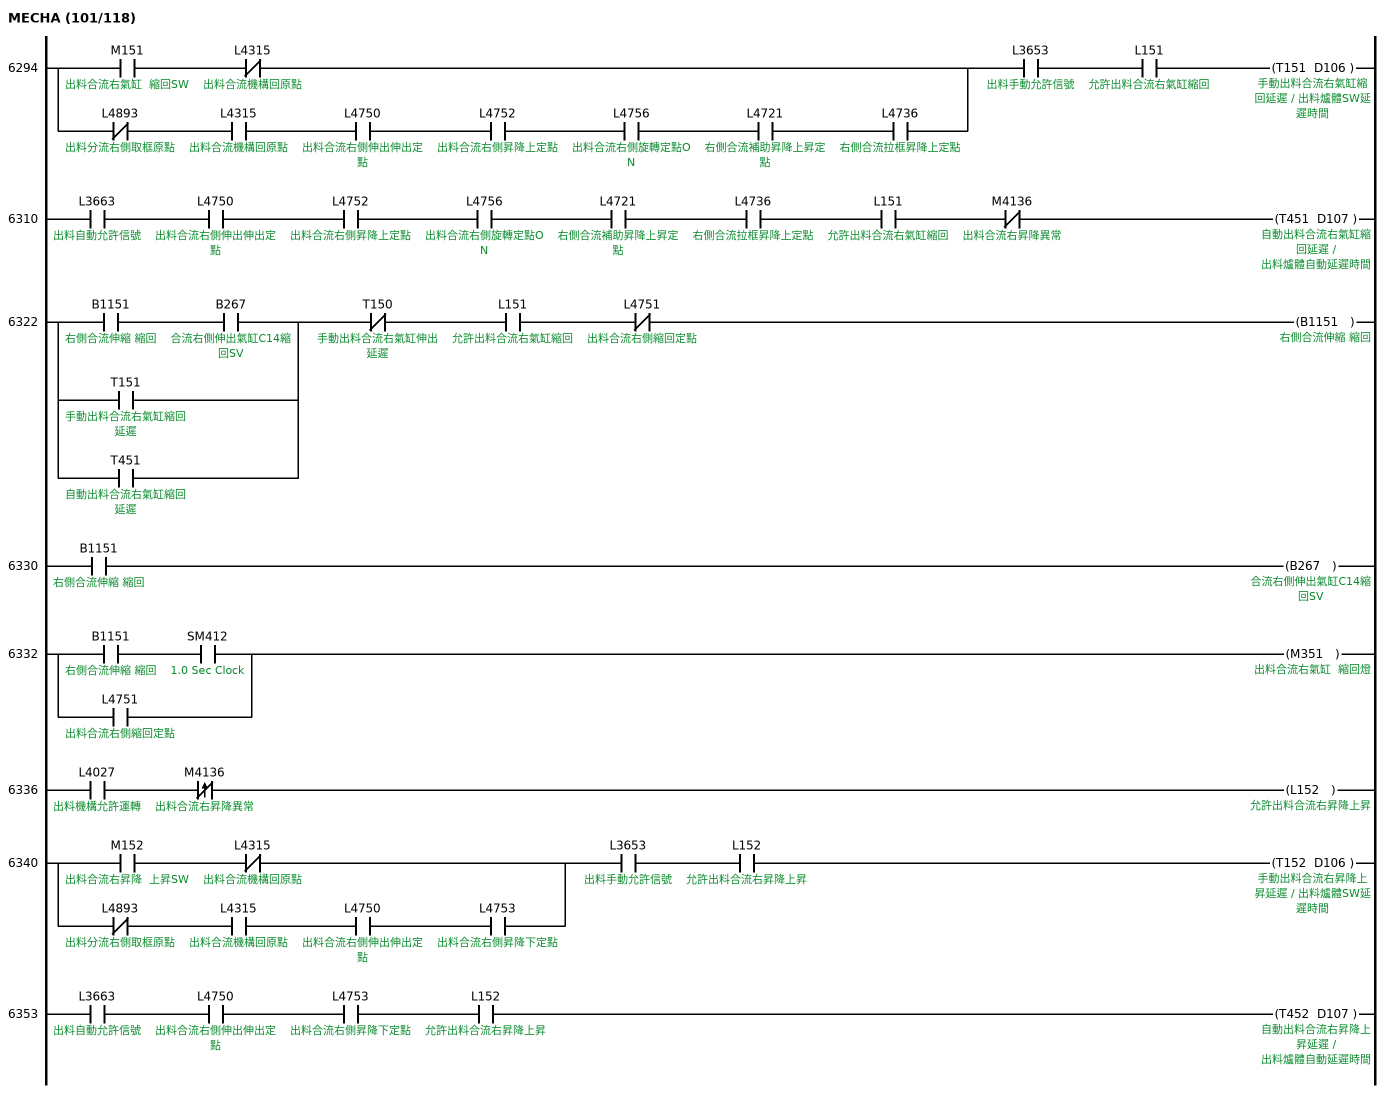
6294  LD      M151  ; 出料合流右氣缸  縮回SW
      ANI     L4315  ; 出料合流機構回原點
      LDI     L4893  ; 出料分流右側取框原點
      AND     L4315  ; 出料合流機構回原點
      AND     L4750  ; 出料合流右側伸出伸出定點
      AND     L4752  ; 出料合流右側昇降上定點
      AND     L4756  ; 出料合流右側旋轉定點ON
      AND     L4721  ; 右側合流補助昇降上昇定點
      AND     L4736  ; 右側合流拉框昇降上定點
      ORB
      AND     L3653  ; 出料手動允許信號
      AND     L151  ; 允許出料合流右氣缸縮回
      OUT     T151 D106  ; 手動出料合流右氣缸縮回延遲 / 出料爐體SW延遲時間
6310  LD      L3663  ; 出料自動允許信號
      AND     L4750  ; 出料合流右側伸出伸出定點
      AND     L4752  ; 出料合流右側昇降上定點
      AND     L4756  ; 出料合流右側旋轉定點ON
      AND     L4721  ; 右側合流補助昇降上昇定點
      AND     L4736  ; 右側合流拉框昇降上定點
      AND     L151  ; 允許出料合流右氣缸縮回
      ANI     M4136  ; 出料合流右昇降異常
      OUT     T451 D107  ; 自動出料合流右氣缸縮回延遲 / 出料爐體自動延遲時間
6322  LD      B1151  ; 右側合流伸縮 縮回
      AND     B267  ; 合流右側伸出氣缸C14縮回SV
      OR      T151  ; 手動出料合流右氣缸縮回延遲
      OR      T451  ; 自動出料合流右氣缸縮回延遲
      ANI     T150  ; 手動出料合流右氣缸伸出延遲
      AND     L151  ; 允許出料合流右氣缸縮回
      ANI     L4751  ; 出料合流右側縮回定點
      OUT     B1151  ; 右側合流伸縮 縮回
6330  LD      B1151  ; 右側合流伸縮 縮回
      OUT     B267  ; 合流右側伸出氣缸C14縮回SV
6332  LD      B1151  ; 右側合流伸縮 縮回
      AND     SM412  ; 1.0 Sec Clock
      OR      L4751  ; 出料合流右側縮回定點
      OUT     M351  ; 出料合流右氣缸  縮回燈
6336  LD      L4027  ; 出料機構允許運轉
      ANDPI   M4136  ; 出料合流右昇降異常
      OUT     L152  ; 允許出料合流右昇降上昇
6340  LD      M152  ; 出料合流右昇降  上昇SW
      ANI     L4315  ; 出料合流機構回原點
      LDI     L4893  ; 出料分流右側取框原點
      AND     L4315  ; 出料合流機構回原點
      AND     L4750  ; 出料合流右側伸出伸出定點
      AND     L4753  ; 出料合流右側昇降下定點
      ORB
      AND     L3653  ; 出料手動允許信號
      AND     L152  ; 允許出料合流右昇降上昇
      OUT     T152 D106  ; 手動出料合流右昇降上昇延遲 / 出料爐體SW延遲時間
6353  LD      L3663  ; 出料自動允許信號
      AND     L4750  ; 出料合流右側伸出伸出定點
      AND     L4753  ; 出料合流右側昇降下定點
      AND     L152  ; 允許出料合流右昇降上昇
      OUT     T452 D107  ; 自動出料合流右昇降上昇延遲 / 出料爐體自動延遲時間
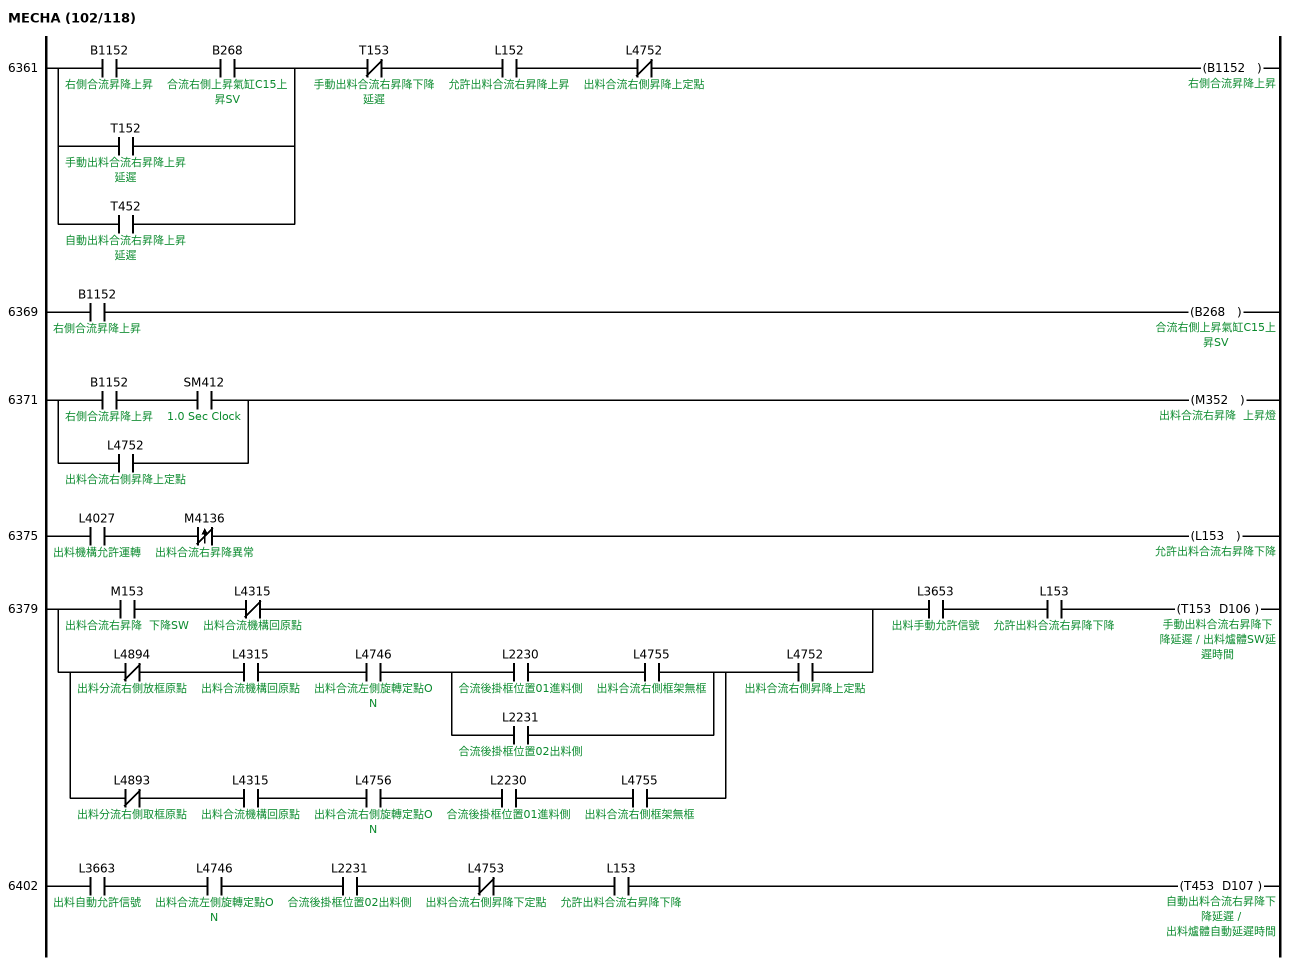
6361  LD      B1152  ; 右側合流昇降上昇
      AND     B268  ; 合流右側上昇氣缸C15上昇SV
      OR      T152  ; 手動出料合流右昇降上昇延遲
      OR      T452  ; 自動出料合流右昇降上昇延遲
      ANI     T153  ; 手動出料合流右昇降下降延遲
      AND     L152  ; 允許出料合流右昇降上昇
      ANI     L4752  ; 出料合流右側昇降上定點
      OUT     B1152  ; 右側合流昇降上昇
6369  LD      B1152  ; 右側合流昇降上昇
      OUT     B268  ; 合流右側上昇氣缸C15上昇SV
6371  LD      B1152  ; 右側合流昇降上昇
      AND     SM412  ; 1.0 Sec Clock
      OR      L4752  ; 出料合流右側昇降上定點
      OUT     M352  ; 出料合流右昇降  上昇燈
6375  LD      L4027  ; 出料機構允許運轉
      ANDPI   M4136  ; 出料合流右昇降異常
      OUT     L153  ; 允許出料合流右昇降下降
6379  LD      M153  ; 出料合流右昇降  下降SW
      ANI     L4315  ; 出料合流機構回原點
      LDI     L4894  ; 出料分流右側放框原點
      AND     L4315  ; 出料合流機構回原點
      AND     L4746  ; 出料合流左側旋轉定點ON
      LD      L2230  ; 合流後掛框位置01進料側
      AND     L4755  ; 出料合流右側框架無框
      OR      L2231  ; 合流後掛框位置02出料側
      ANB
      LDI     L4893  ; 出料分流右側取框原點
      AND     L4315  ; 出料合流機構回原點
      AND     L4756  ; 出料合流右側旋轉定點ON
      AND     L2230  ; 合流後掛框位置01進料側
      AND     L4755  ; 出料合流右側框架無框
      ORB
      AND     L4752  ; 出料合流右側昇降上定點
      ORB
      AND     L3653  ; 出料手動允許信號
      AND     L153  ; 允許出料合流右昇降下降
      OUT     T153 D106  ; 手動出料合流右昇降下降延遲 / 出料爐體SW延遲時間
6402  LD      L3663  ; 出料自動允許信號
      AND     L4746  ; 出料合流左側旋轉定點ON
      AND     L2231  ; 合流後掛框位置02出料側
      ANI     L4753  ; 出料合流右側昇降下定點
      AND     L153  ; 允許出料合流右昇降下降
      OUT     T453 D107  ; 自動出料合流右昇降下降延遲 / 出料爐體自動延遲時間
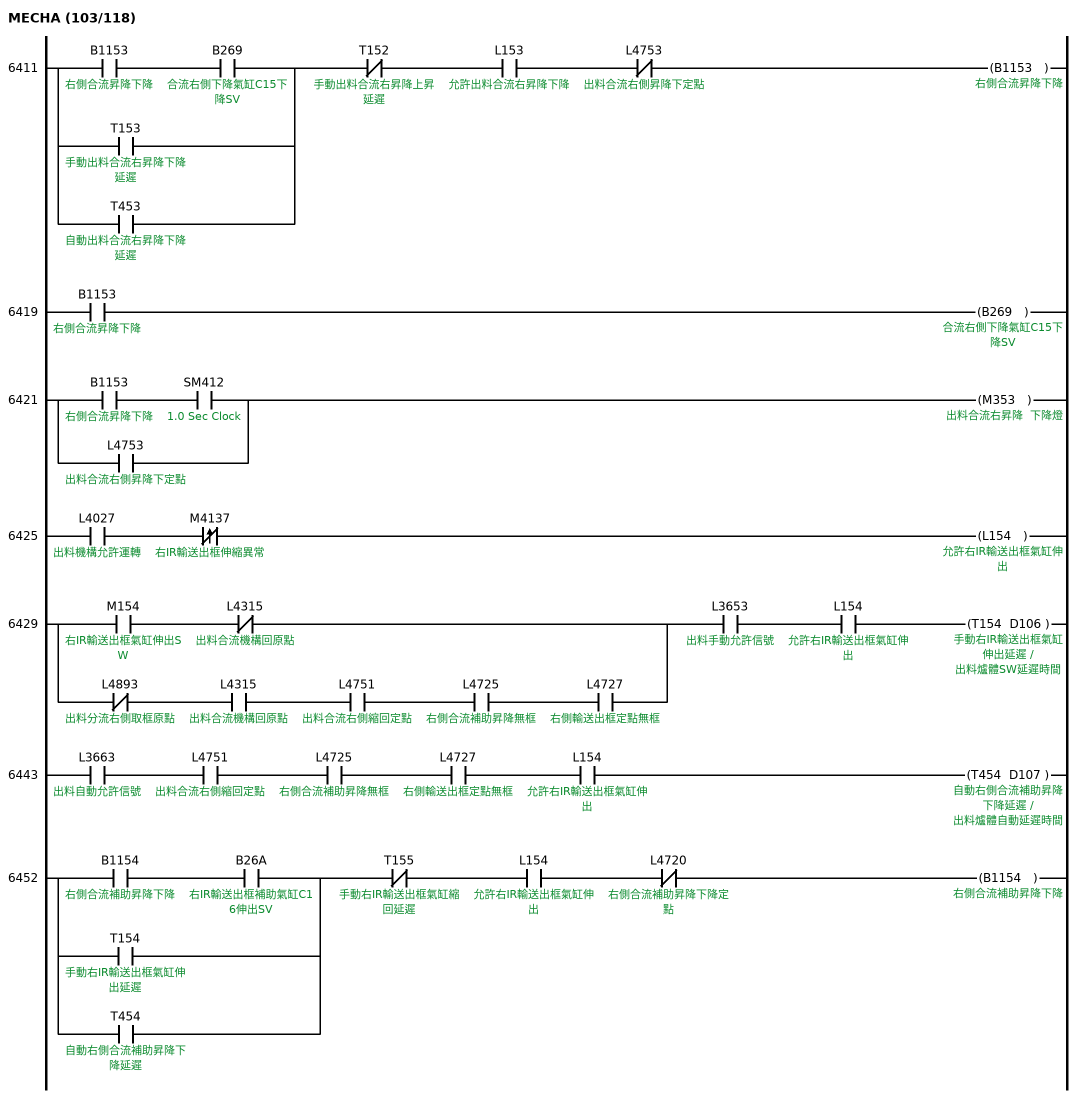
6411  LD      B1153  ; 右側合流昇降下降
      AND     B269  ; 合流右側下降氣缸C15下降SV
      OR      T153  ; 手動出料合流右昇降下降延遲
      OR      T453  ; 自動出料合流右昇降下降延遲
      ANI     T152  ; 手動出料合流右昇降上昇延遲
      AND     L153  ; 允許出料合流右昇降下降
      ANI     L4753  ; 出料合流右側昇降下定點
      OUT     B1153  ; 右側合流昇降下降
6419  LD      B1153  ; 右側合流昇降下降
      OUT     B269  ; 合流右側下降氣缸C15下降SV
6421  LD      B1153  ; 右側合流昇降下降
      AND     SM412  ; 1.0 Sec Clock
      OR      L4753  ; 出料合流右側昇降下定點
      OUT     M353  ; 出料合流右昇降  下降燈
6425  LD      L4027  ; 出料機構允許運轉
      ANDPI   M4137  ; 右IR輸送出框伸縮異常
      OUT     L154  ; 允許右IR輸送出框氣缸伸出
6429  LD      M154  ; 右IR輸送出框氣缸伸出SW
      ANI     L4315  ; 出料合流機構回原點
      LDI     L4893  ; 出料分流右側取框原點
      AND     L4315  ; 出料合流機構回原點
      AND     L4751  ; 出料合流右側縮回定點
      AND     L4725  ; 右側合流補助昇降無框
      AND     L4727  ; 右側輸送出框定點無框
      ORB
      AND     L3653  ; 出料手動允許信號
      AND     L154  ; 允許右IR輸送出框氣缸伸出
      OUT     T154 D106  ; 手動右IR輸送出框氣缸伸出延遲 / 出料爐體SW延遲時間
6443  LD      L3663  ; 出料自動允許信號
      AND     L4751  ; 出料合流右側縮回定點
      AND     L4725  ; 右側合流補助昇降無框
      AND     L4727  ; 右側輸送出框定點無框
      AND     L154  ; 允許右IR輸送出框氣缸伸出
      OUT     T454 D107  ; 自動右側合流補助昇降下降延遲 / 出料爐體自動延遲時間
6452  LD      B1154  ; 右側合流補助昇降下降
      AND     B26A  ; 右IR輸送出框補助氣缸C16伸出SV
      OR      T154  ; 手動右IR輸送出框氣缸伸出延遲
      OR      T454  ; 自動右側合流補助昇降下降延遲
      ANI     T155  ; 手動右IR輸送出框氣缸縮回延遲
      AND     L154  ; 允許右IR輸送出框氣缸伸出
      ANI     L4720  ; 右側合流補助昇降下降定點
      OUT     B1154  ; 右側合流補助昇降下降
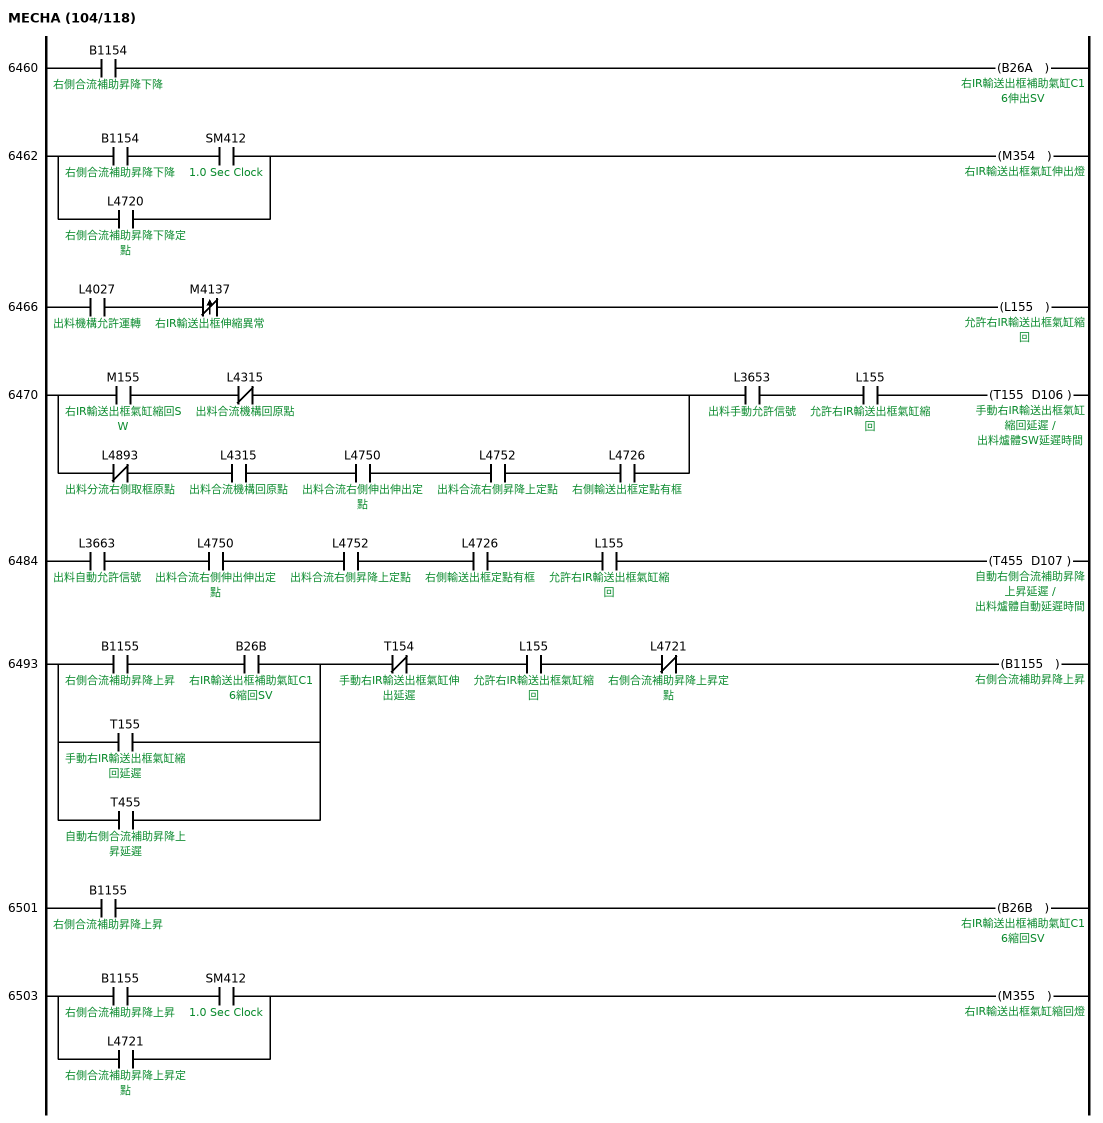
6460  LD      B1154  ; 右側合流補助昇降下降
      OUT     B26A  ; 右IR輸送出框補助氣缸C16伸出SV
6462  LD      B1154  ; 右側合流補助昇降下降
      AND     SM412  ; 1.0 Sec Clock
      OR      L4720  ; 右側合流補助昇降下降定點
      OUT     M354  ; 右IR輸送出框氣缸伸出燈
6466  LD      L4027  ; 出料機構允許運轉
      ANDPI   M4137  ; 右IR輸送出框伸縮異常
      OUT     L155  ; 允許右IR輸送出框氣缸縮回
6470  LD      M155  ; 右IR輸送出框氣缸縮回SW
      ANI     L4315  ; 出料合流機構回原點
      LDI     L4893  ; 出料分流右側取框原點
      AND     L4315  ; 出料合流機構回原點
      AND     L4750  ; 出料合流右側伸出伸出定點
      AND     L4752  ; 出料合流右側昇降上定點
      AND     L4726  ; 右側輸送出框定點有框
      ORB
      AND     L3653  ; 出料手動允許信號
      AND     L155  ; 允許右IR輸送出框氣缸縮回
      OUT     T155 D106  ; 手動右IR輸送出框氣缸縮回延遲 / 出料爐體SW延遲時間
6484  LD      L3663  ; 出料自動允許信號
      AND     L4750  ; 出料合流右側伸出伸出定點
      AND     L4752  ; 出料合流右側昇降上定點
      AND     L4726  ; 右側輸送出框定點有框
      AND     L155  ; 允許右IR輸送出框氣缸縮回
      OUT     T455 D107  ; 自動右側合流補助昇降上昇延遲 / 出料爐體自動延遲時間
6493  LD      B1155  ; 右側合流補助昇降上昇
      AND     B26B  ; 右IR輸送出框補助氣缸C16縮回SV
      OR      T155  ; 手動右IR輸送出框氣缸縮回延遲
      OR      T455  ; 自動右側合流補助昇降上昇延遲
      ANI     T154  ; 手動右IR輸送出框氣缸伸出延遲
      AND     L155  ; 允許右IR輸送出框氣缸縮回
      ANI     L4721  ; 右側合流補助昇降上昇定點
      OUT     B1155  ; 右側合流補助昇降上昇
6501  LD      B1155  ; 右側合流補助昇降上昇
      OUT     B26B  ; 右IR輸送出框補助氣缸C16縮回SV
6503  LD      B1155  ; 右側合流補助昇降上昇
      AND     SM412  ; 1.0 Sec Clock
      OR      L4721  ; 右側合流補助昇降上昇定點
      OUT     M355  ; 右IR輸送出框氣缸縮回燈
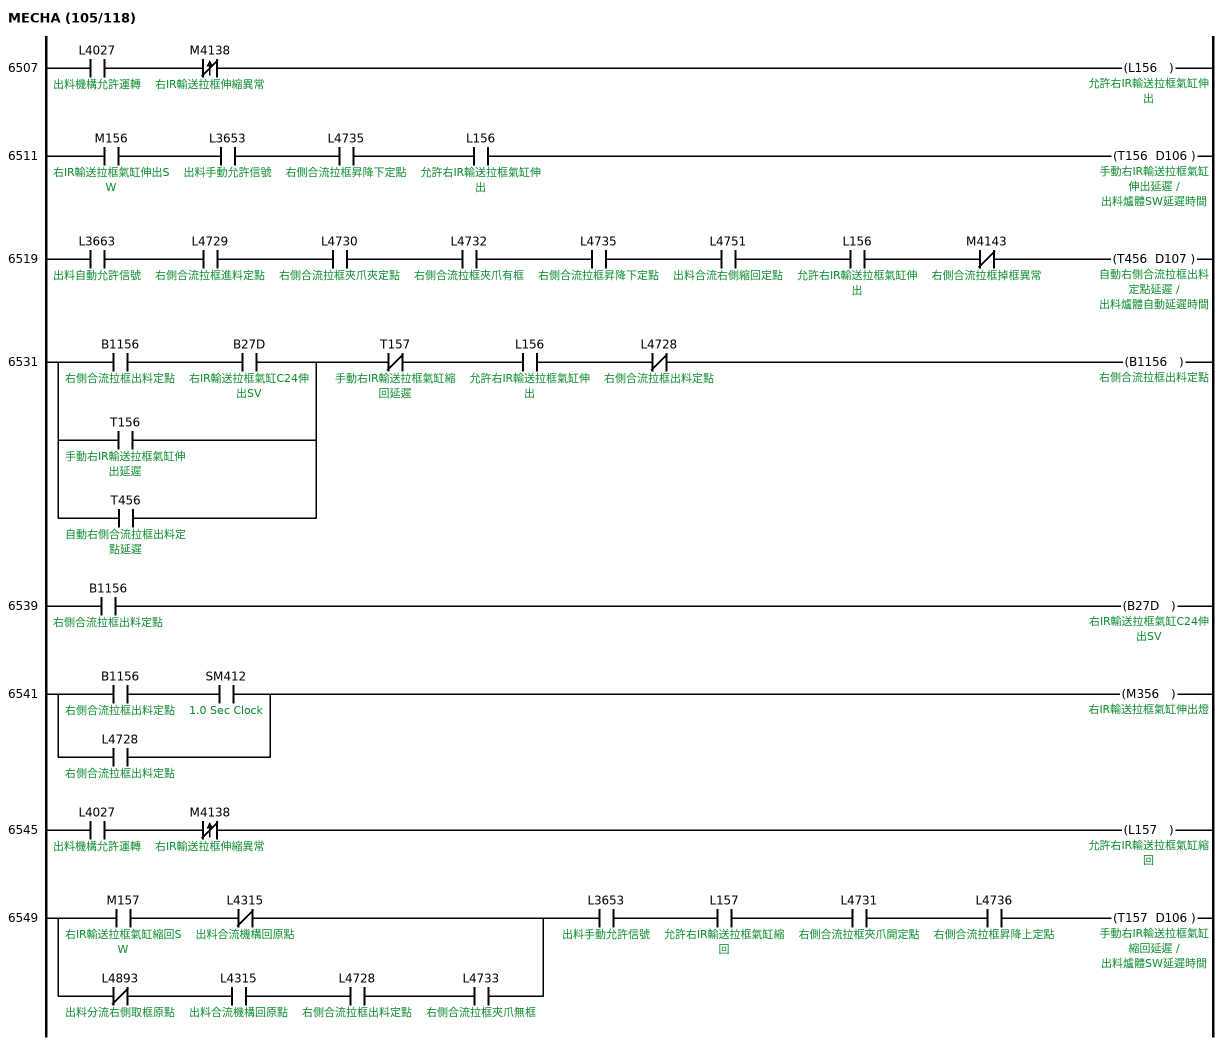
6507  LD      L4027  ; 出料機構允許運轉
      ANDPI   M4138  ; 右IR輸送拉框伸縮異常
      OUT     L156  ; 允許右IR輸送拉框氣缸伸出
6511  LD      M156  ; 右IR輸送拉框氣缸伸出SW
      AND     L3653  ; 出料手動允許信號
      AND     L4735  ; 右側合流拉框昇降下定點
      AND     L156  ; 允許右IR輸送拉框氣缸伸出
      OUT     T156 D106  ; 手動右IR輸送拉框氣缸伸出延遲 / 出料爐體SW延遲時間
6519  LD      L3663  ; 出料自動允許信號
      AND     L4729  ; 右側合流拉框進料定點
      AND     L4730  ; 右側合流拉框夾爪夾定點
      AND     L4732  ; 右側合流拉框夾爪有框
      AND     L4735  ; 右側合流拉框昇降下定點
      AND     L4751  ; 出料合流右側縮回定點
      AND     L156  ; 允許右IR輸送拉框氣缸伸出
      ANI     M4143  ; 右側合流拉框掉框異常
      OUT     T456 D107  ; 自動右側合流拉框出料定點延遲 / 出料爐體自動延遲時間
6531  LD      B1156  ; 右側合流拉框出料定點
      AND     B27D  ; 右IR輸送拉框氣缸C24伸出SV
      OR      T156  ; 手動右IR輸送拉框氣缸伸出延遲
      OR      T456  ; 自動右側合流拉框出料定點延遲
      ANI     T157  ; 手動右IR輸送拉框氣缸縮回延遲
      AND     L156  ; 允許右IR輸送拉框氣缸伸出
      ANI     L4728  ; 右側合流拉框出料定點
      OUT     B1156  ; 右側合流拉框出料定點
6539  LD      B1156  ; 右側合流拉框出料定點
      OUT     B27D  ; 右IR輸送拉框氣缸C24伸出SV
6541  LD      B1156  ; 右側合流拉框出料定點
      AND     SM412  ; 1.0 Sec Clock
      OR      L4728  ; 右側合流拉框出料定點
      OUT     M356  ; 右IR輸送拉框氣缸伸出燈
6545  LD      L4027  ; 出料機構允許運轉
      ANDPI   M4138  ; 右IR輸送拉框伸縮異常
      OUT     L157  ; 允許右IR輸送拉框氣缸縮回
6549  LD      M157  ; 右IR輸送拉框氣缸縮回SW
      ANI     L4315  ; 出料合流機構回原點
      LDI     L4893  ; 出料分流右側取框原點
      AND     L4315  ; 出料合流機構回原點
      AND     L4728  ; 右側合流拉框出料定點
      AND     L4733  ; 右側合流拉框夾爪無框
      ORB
      AND     L3653  ; 出料手動允許信號
      AND     L157  ; 允許右IR輸送拉框氣缸縮回
      AND     L4731  ; 右側合流拉框夾爪開定點
      AND     L4736  ; 右側合流拉框昇降上定點
      OUT     T157 D106  ; 手動右IR輸送拉框氣缸縮回延遲 / 出料爐體SW延遲時間
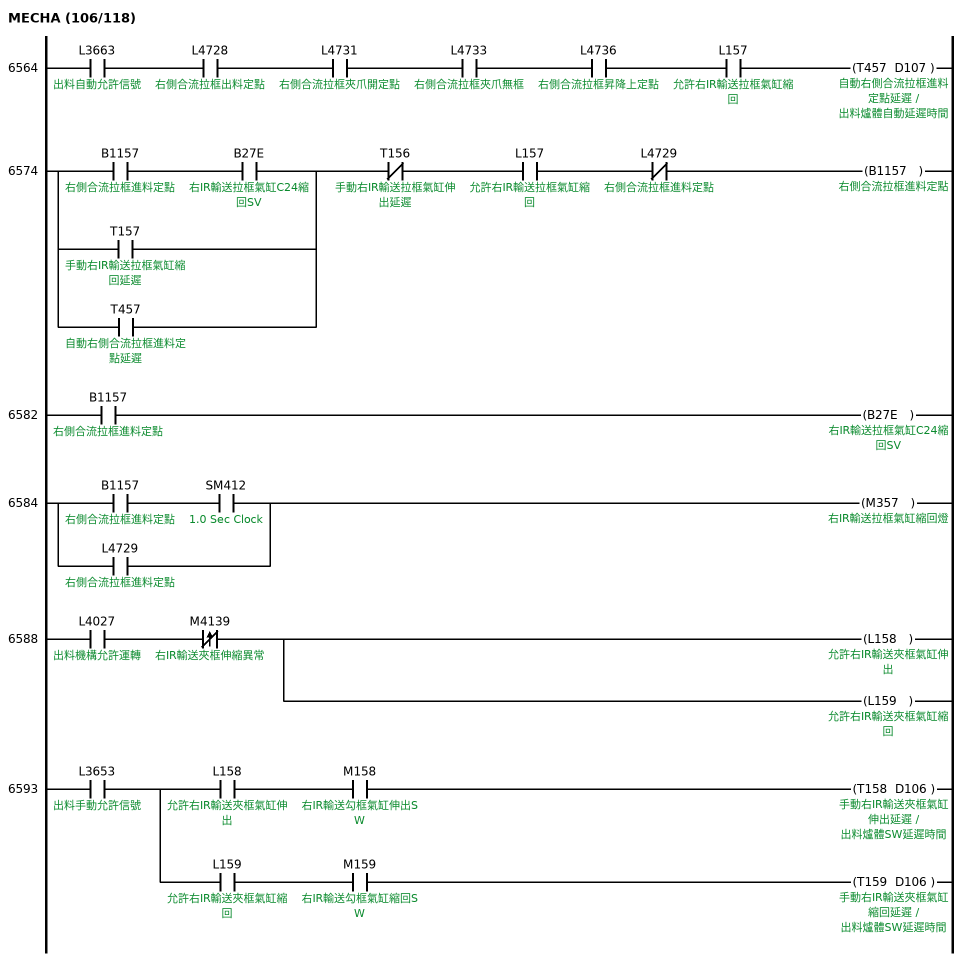
6564  LD      L3663  ; 出料自動允許信號
      AND     L4728  ; 右側合流拉框出料定點
      AND     L4731  ; 右側合流拉框夾爪開定點
      AND     L4733  ; 右側合流拉框夾爪無框
      AND     L4736  ; 右側合流拉框昇降上定點
      AND     L157  ; 允許右IR輸送拉框氣缸縮回
      OUT     T457 D107  ; 自動右側合流拉框進料定點延遲 / 出料爐體自動延遲時間
6574  LD      B1157  ; 右側合流拉框進料定點
      AND     B27E  ; 右IR輸送拉框氣缸C24縮回SV
      OR      T157  ; 手動右IR輸送拉框氣缸縮回延遲
      OR      T457  ; 自動右側合流拉框進料定點延遲
      ANI     T156  ; 手動右IR輸送拉框氣缸伸出延遲
      AND     L157  ; 允許右IR輸送拉框氣缸縮回
      ANI     L4729  ; 右側合流拉框進料定點
      OUT     B1157  ; 右側合流拉框進料定點
6582  LD      B1157  ; 右側合流拉框進料定點
      OUT     B27E  ; 右IR輸送拉框氣缸C24縮回SV
6584  LD      B1157  ; 右側合流拉框進料定點
      AND     SM412  ; 1.0 Sec Clock
      OR      L4729  ; 右側合流拉框進料定點
      OUT     M357  ; 右IR輸送拉框氣缸縮回燈
6588  LD      L4027  ; 出料機構允許運轉
      ANDPI   M4139  ; 右IR輸送夾框伸縮異常
      OUT     L158  ; 允許右IR輸送夾框氣缸伸出
      OUT     L159  ; 允許右IR輸送夾框氣缸縮回
6593  LD      L3653  ; 出料手動允許信號
      MPS
      AND     L158  ; 允許右IR輸送夾框氣缸伸出
      AND     M158  ; 右IR輸送勾框氣缸伸出SW
      OUT     T158 D106  ; 手動右IR輸送夾框氣缸伸出延遲 / 出料爐體SW延遲時間
      MPP
      AND     L159  ; 允許右IR輸送夾框氣缸縮回
      AND     M159  ; 右IR輸送勾框氣缸縮回SW
      OUT     T159 D106  ; 手動右IR輸送夾框氣缸縮回延遲 / 出料爐體SW延遲時間
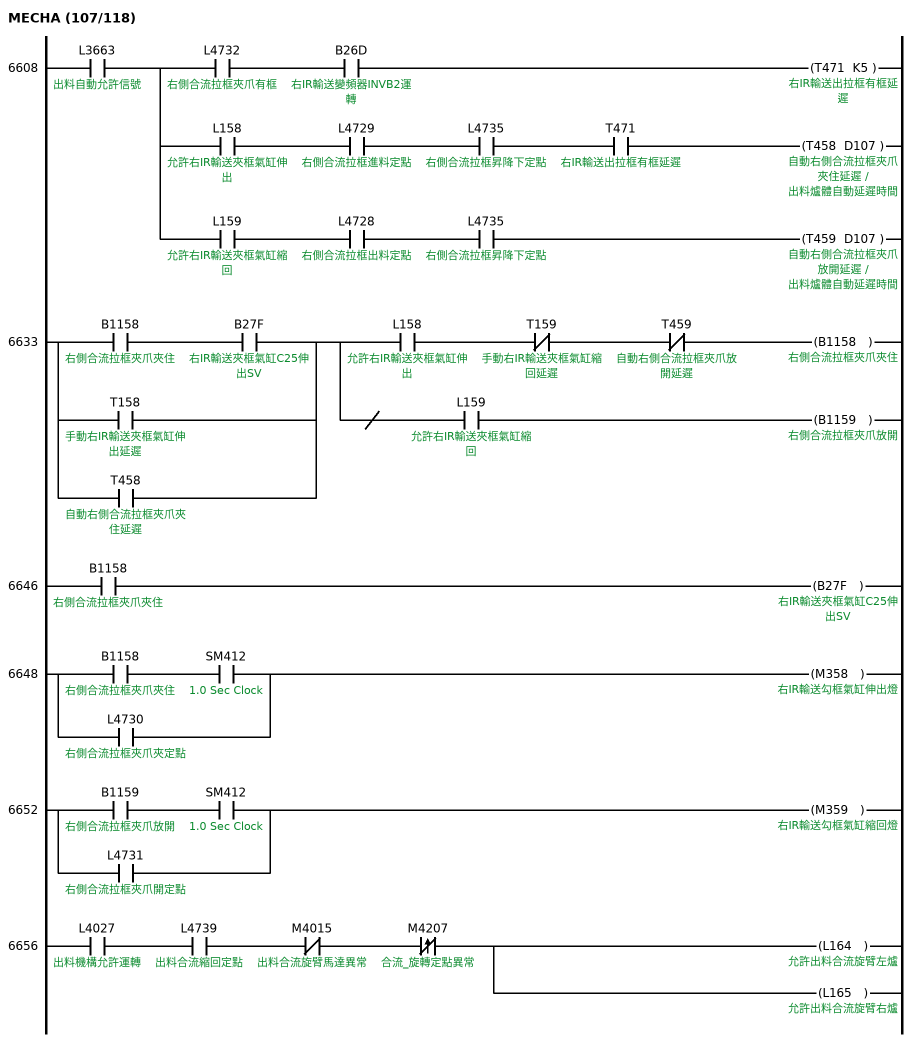
6608  LD      L3663  ; 出料自動允許信號
      MPS
      AND     L4732  ; 右側合流拉框夾爪有框
      AND     B26D  ; 右IR輸送變頻器INVB2運轉
      OUT     T471 K5  ; 右IR輸送出拉框有框延遲
      MRD
      AND     L158  ; 允許右IR輸送夾框氣缸伸出
      AND     L4729  ; 右側合流拉框進料定點
      AND     L4735  ; 右側合流拉框昇降下定點
      AND     T471  ; 右IR輸送出拉框有框延遲
      OUT     T458 D107  ; 自動右側合流拉框夾爪夾住延遲 / 出料爐體自動延遲時間
      MPP
      AND     L159  ; 允許右IR輸送夾框氣缸縮回
      AND     L4728  ; 右側合流拉框出料定點
      AND     L4735  ; 右側合流拉框昇降下定點
      OUT     T459 D107  ; 自動右側合流拉框夾爪放開延遲 / 出料爐體自動延遲時間
6633  LD      B1158  ; 右側合流拉框夾爪夾住
      AND     B27F  ; 右IR輸送夾框氣缸C25伸出SV
      OR      T158  ; 手動右IR輸送夾框氣缸伸出延遲
      OR      T458  ; 自動右側合流拉框夾爪夾住延遲
      MPS
      AND     L158  ; 允許右IR輸送夾框氣缸伸出
      ANI     T159  ; 手動右IR輸送夾框氣缸縮回延遲
      ANI     T459  ; 自動右側合流拉框夾爪放開延遲
      OUT     B1158  ; 右側合流拉框夾爪夾住
      MPP
      INV
      AND     L159  ; 允許右IR輸送夾框氣缸縮回
      OUT     B1159  ; 右側合流拉框夾爪放開
6646  LD      B1158  ; 右側合流拉框夾爪夾住
      OUT     B27F  ; 右IR輸送夾框氣缸C25伸出SV
6648  LD      B1158  ; 右側合流拉框夾爪夾住
      AND     SM412  ; 1.0 Sec Clock
      OR      L4730  ; 右側合流拉框夾爪夾定點
      OUT     M358  ; 右IR輸送勾框氣缸伸出燈
6652  LD      B1159  ; 右側合流拉框夾爪放開
      AND     SM412  ; 1.0 Sec Clock
      OR      L4731  ; 右側合流拉框夾爪開定點
      OUT     M359  ; 右IR輸送勾框氣缸縮回燈
6656  LD      L4027  ; 出料機構允許運轉
      AND     L4739  ; 出料合流縮回定點
      ANI     M4015  ; 出料合流旋臂馬達異常
      ANDPI   M4207  ; 合流_旋轉定點異常
      OUT     L164  ; 允許出料合流旋臂左爐
      OUT     L165  ; 允許出料合流旋臂右爐
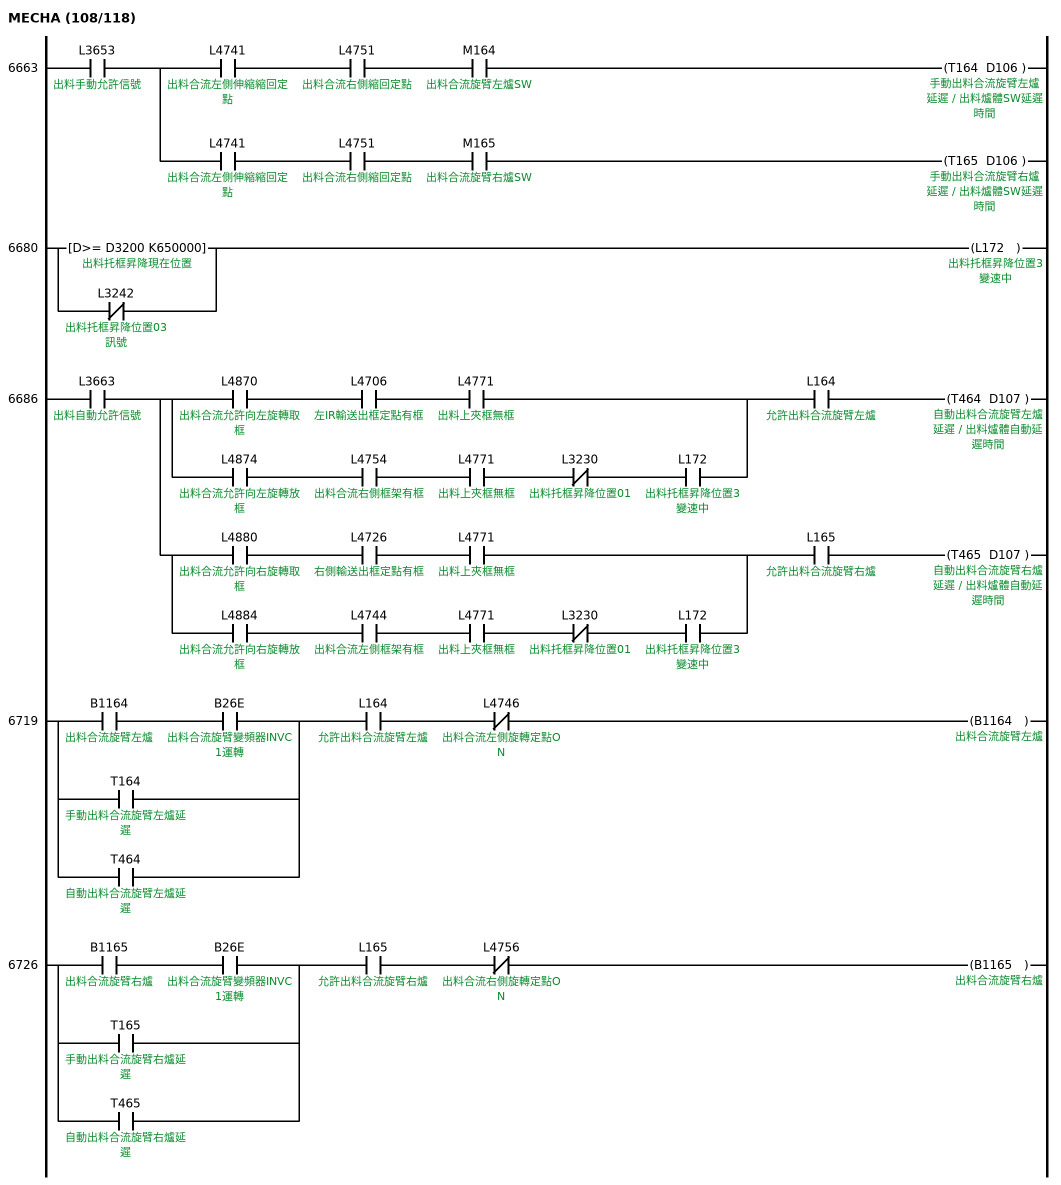
6663  LD      L3653  ; 出料手動允許信號
      MPS
      AND     L4741  ; 出料合流左側伸縮縮回定點
      AND     L4751  ; 出料合流右側縮回定點
      AND     M164  ; 出料合流旋臂左爐SW
      OUT     T164 D106  ; 手動出料合流旋臂左爐延遲 / 出料爐體SW延遲時間
      MPP
      AND     L4741  ; 出料合流左側伸縮縮回定點
      AND     L4751  ; 出料合流右側縮回定點
      AND     M165  ; 出料合流旋臂右爐SW
      OUT     T165 D106  ; 手動出料合流旋臂右爐延遲 / 出料爐體SW延遲時間
6680  LDD>=   D3200 K650000  ; 出料托框昇降現在位置
      ORI     L3242  ; 出料托框昇降位置03 訊號
      OUT     L172  ; 出料托框昇降位置3 變速中
6686  LD      L3663  ; 出料自動允許信號
      MPS
      LD      L4870  ; 出料合流允許向左旋轉取框
      AND     L4706  ; 左IR輸送出框定點有框
      AND     L4771  ; 出料上夾框無框
      LD      L4874  ; 出料合流允許向左旋轉放框
      AND     L4754  ; 出料合流右側框架有框
      AND     L4771  ; 出料上夾框無框
      ANI     L3230  ; 出料托框昇降位置01
      AND     L172  ; 出料托框昇降位置3 變速中
      ORB
      ANB
      AND     L164  ; 允許出料合流旋臂左爐
      OUT     T464 D107  ; 自動出料合流旋臂左爐延遲 / 出料爐體自動延遲時間
      MPP
      LD      L4880  ; 出料合流允許向右旋轉取框
      AND     L4726  ; 右側輸送出框定點有框
      AND     L4771  ; 出料上夾框無框
      LD      L4884  ; 出料合流允許向右旋轉放框
      AND     L4744  ; 出料合流左側框架有框
      AND     L4771  ; 出料上夾框無框
      ANI     L3230  ; 出料托框昇降位置01
      AND     L172  ; 出料托框昇降位置3 變速中
      ORB
      ANB
      AND     L165  ; 允許出料合流旋臂右爐
      OUT     T465 D107  ; 自動出料合流旋臂右爐延遲 / 出料爐體自動延遲時間
6719  LD      B1164  ; 出料合流旋臂左爐
      AND     B26E  ; 出料合流旋臂變頻器INVC1運轉
      OR      T164  ; 手動出料合流旋臂左爐延遲
      OR      T464  ; 自動出料合流旋臂左爐延遲
      AND     L164  ; 允許出料合流旋臂左爐
      ANI     L4746  ; 出料合流左側旋轉定點ON
      OUT     B1164  ; 出料合流旋臂左爐
6726  LD      B1165  ; 出料合流旋臂右爐
      AND     B26E  ; 出料合流旋臂變頻器INVC1運轉
      OR      T165  ; 手動出料合流旋臂右爐延遲
      OR      T465  ; 自動出料合流旋臂右爐延遲
      AND     L165  ; 允許出料合流旋臂右爐
      ANI     L4756  ; 出料合流右側旋轉定點ON
      OUT     B1165  ; 出料合流旋臂右爐
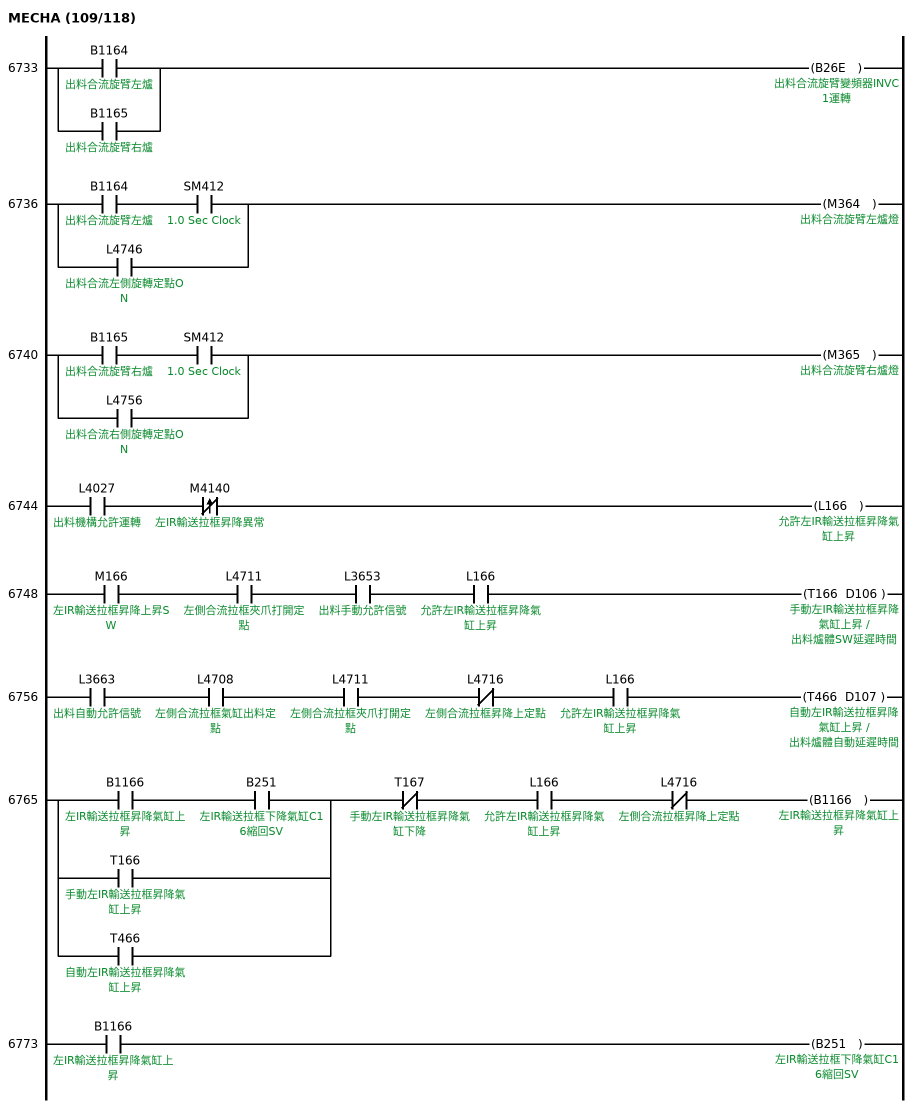
6733  LD      B1164  ; 出料合流旋臂左爐
      OR      B1165  ; 出料合流旋臂右爐
      OUT     B26E  ; 出料合流旋臂變頻器INVC1運轉
6736  LD      B1164  ; 出料合流旋臂左爐
      AND     SM412  ; 1.0 Sec Clock
      OR      L4746  ; 出料合流左側旋轉定點ON
      OUT     M364  ; 出料合流旋臂左爐燈
6740  LD      B1165  ; 出料合流旋臂右爐
      AND     SM412  ; 1.0 Sec Clock
      OR      L4756  ; 出料合流右側旋轉定點ON
      OUT     M365  ; 出料合流旋臂右爐燈
6744  LD      L4027  ; 出料機構允許運轉
      ANDPI   M4140  ; 左IR輸送拉框昇降異常
      OUT     L166  ; 允許左IR輸送拉框昇降氣缸上昇
6748  LD      M166  ; 左IR輸送拉框昇降上昇SW
      AND     L4711  ; 左側合流拉框夾爪打開定點
      AND     L3653  ; 出料手動允許信號
      AND     L166  ; 允許左IR輸送拉框昇降氣缸上昇
      OUT     T166 D106  ; 手動左IR輸送拉框昇降氣缸上昇 / 出料爐體SW延遲時間
6756  LD      L3663  ; 出料自動允許信號
      AND     L4708  ; 左側合流拉框氣缸出料定點
      AND     L4711  ; 左側合流拉框夾爪打開定點
      ANI     L4716  ; 左側合流拉框昇降上定點
      AND     L166  ; 允許左IR輸送拉框昇降氣缸上昇
      OUT     T466 D107  ; 自動左IR輸送拉框昇降氣缸上昇 / 出料爐體自動延遲時間
6765  LD      B1166  ; 左IR輸送拉框昇降氣缸上昇
      AND     B251  ; 左IR輸送拉框下降氣缸C16縮回SV
      OR      T166  ; 手動左IR輸送拉框昇降氣缸上昇
      OR      T466  ; 自動左IR輸送拉框昇降氣缸上昇
      ANI     T167  ; 手動左IR輸送拉框昇降氣缸下降
      AND     L166  ; 允許左IR輸送拉框昇降氣缸上昇
      ANI     L4716  ; 左側合流拉框昇降上定點
      OUT     B1166  ; 左IR輸送拉框昇降氣缸上昇
6773  LD      B1166  ; 左IR輸送拉框昇降氣缸上昇
      OUT     B251  ; 左IR輸送拉框下降氣缸C16縮回SV
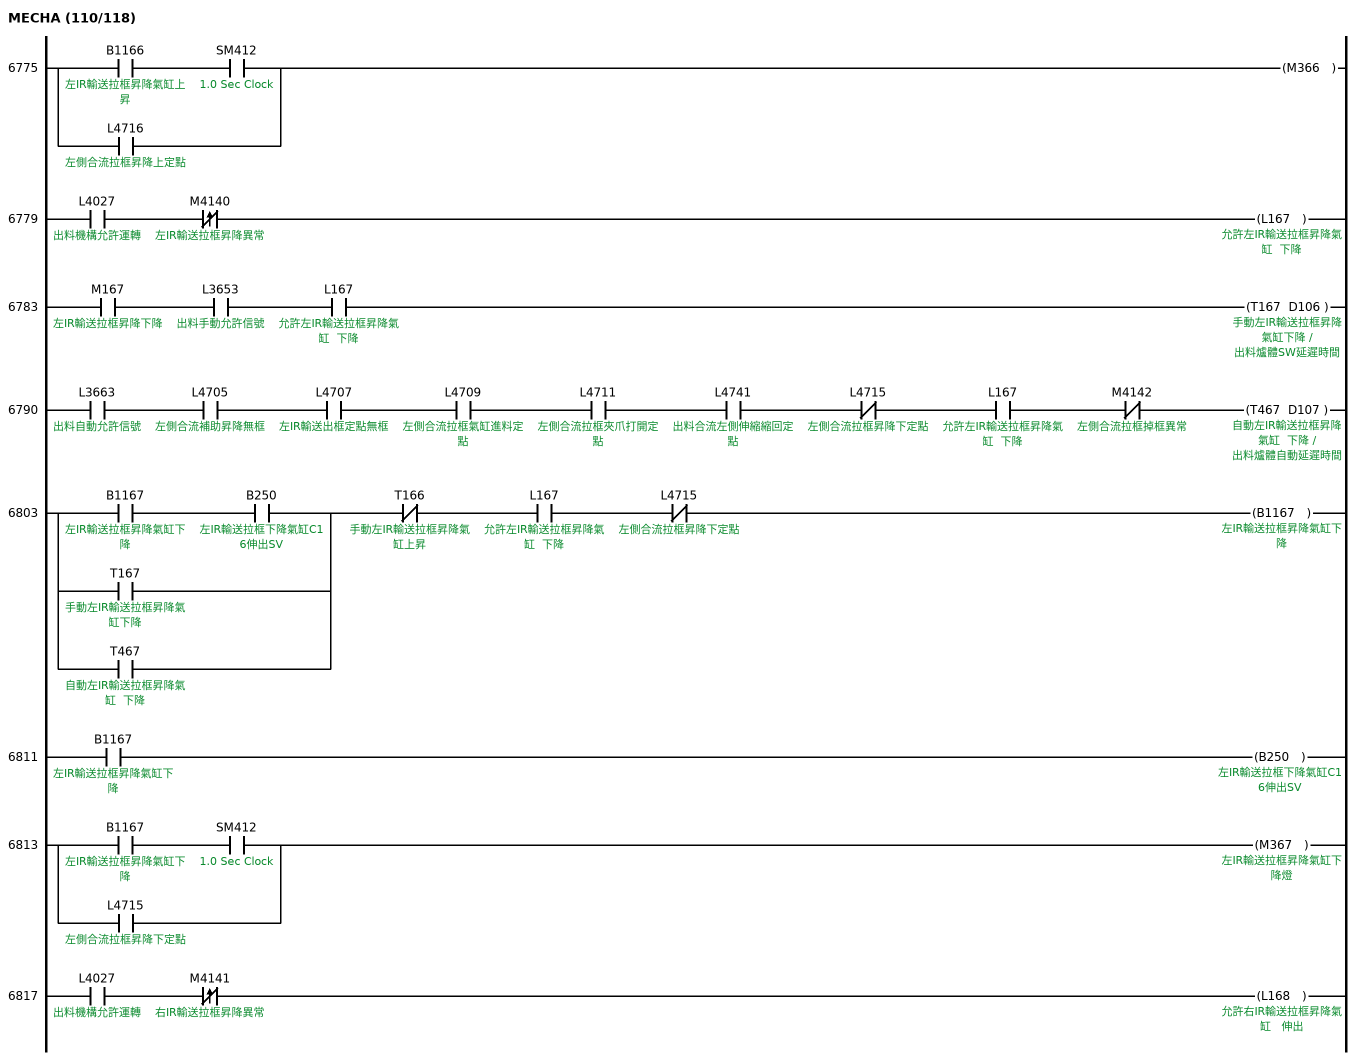
6775  LD      B1166  ; 左IR輸送拉框昇降氣缸上昇
      AND     SM412  ; 1.0 Sec Clock
      OR      L4716  ; 左側合流拉框昇降上定點
      OUT     M366
6779  LD      L4027  ; 出料機構允許運轉
      ANDPI   M4140  ; 左IR輸送拉框昇降異常
      OUT     L167  ; 允許左IR輸送拉框昇降氣缸  下降
6783  LD      M167  ; 左IR輸送拉框昇降下降
      AND     L3653  ; 出料手動允許信號
      AND     L167  ; 允許左IR輸送拉框昇降氣缸  下降
      OUT     T167 D106  ; 手動左IR輸送拉框昇降氣缸下降 / 出料爐體SW延遲時間
6790  LD      L3663  ; 出料自動允許信號
      AND     L4705  ; 左側合流補助昇降無框
      AND     L4707  ; 左IR輸送出框定點無框
      AND     L4709  ; 左側合流拉框氣缸進料定點
      AND     L4711  ; 左側合流拉框夾爪打開定點
      AND     L4741  ; 出料合流左側伸縮縮回定點
      ANI     L4715  ; 左側合流拉框昇降下定點
      AND     L167  ; 允許左IR輸送拉框昇降氣缸  下降
      ANI     M4142  ; 左側合流拉框掉框異常
      OUT     T467 D107  ; 自動左IR輸送拉框昇降氣缸  下降 / 出料爐體自動延遲時間
6803  LD      B1167  ; 左IR輸送拉框昇降氣缸下降
      AND     B250  ; 左IR輸送拉框下降氣缸C16伸出SV
      OR      T167  ; 手動左IR輸送拉框昇降氣缸下降
      OR      T467  ; 自動左IR輸送拉框昇降氣缸  下降
      ANI     T166  ; 手動左IR輸送拉框昇降氣缸上昇
      AND     L167  ; 允許左IR輸送拉框昇降氣缸  下降
      ANI     L4715  ; 左側合流拉框昇降下定點
      OUT     B1167  ; 左IR輸送拉框昇降氣缸下降
6811  LD      B1167  ; 左IR輸送拉框昇降氣缸下降
      OUT     B250  ; 左IR輸送拉框下降氣缸C16伸出SV
6813  LD      B1167  ; 左IR輸送拉框昇降氣缸下降
      AND     SM412  ; 1.0 Sec Clock
      OR      L4715  ; 左側合流拉框昇降下定點
      OUT     M367  ; 左IR輸送拉框昇降氣缸下降燈
6817  LD      L4027  ; 出料機構允許運轉
      ANDPI   M4141  ; 右IR輸送拉框昇降異常
      OUT     L168  ; 允許右IR輸送拉框昇降氣缸   伸出
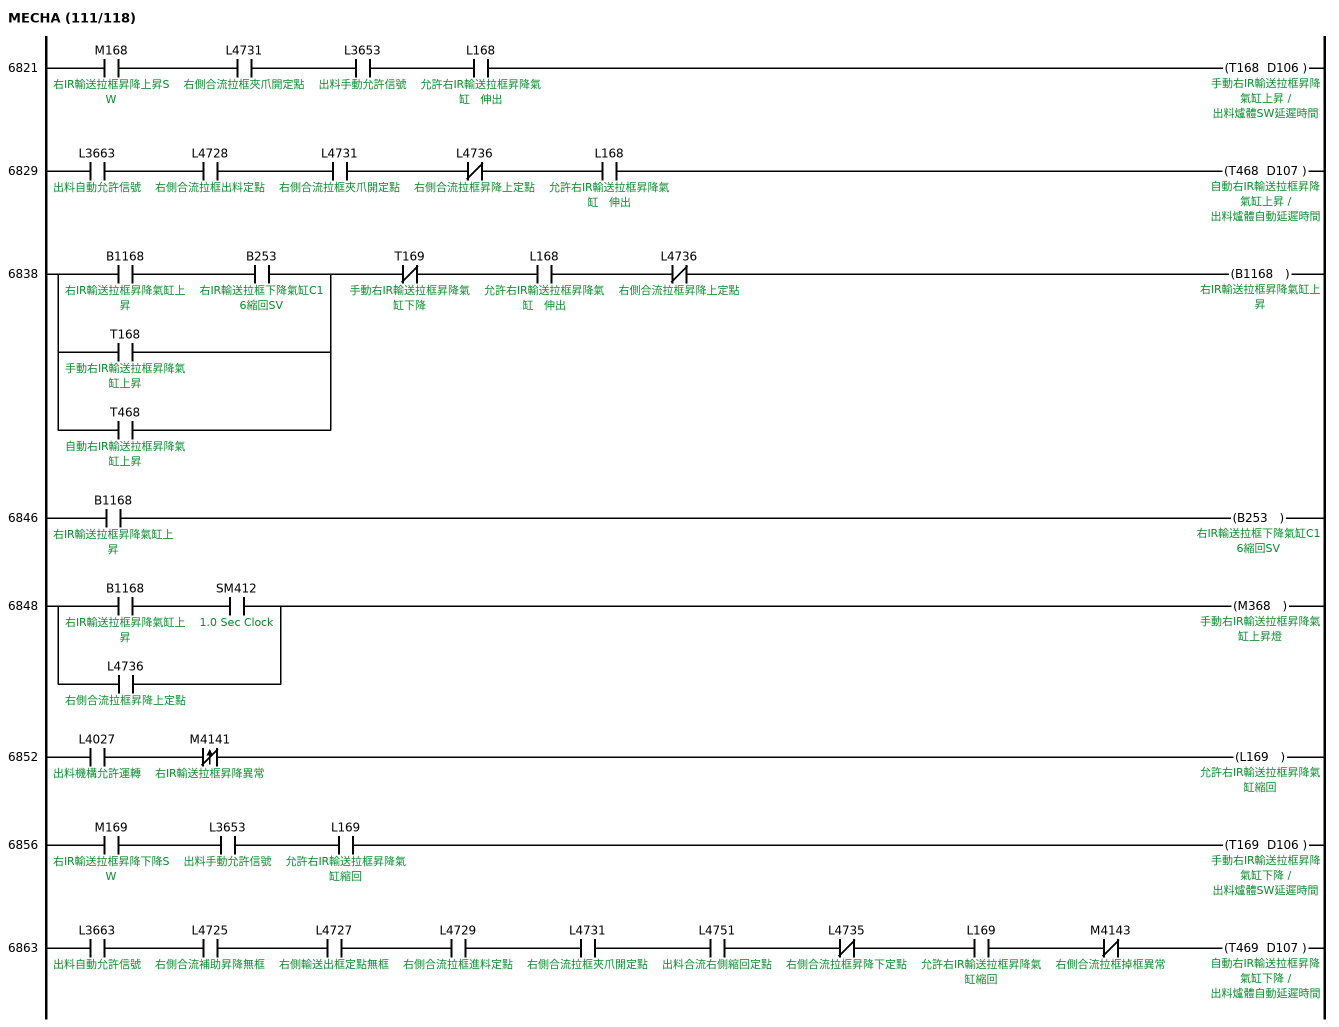
6821  LD      M168  ; 右IR輸送拉框昇降上昇SW
      AND     L4731  ; 右側合流拉框夾爪開定點
      AND     L3653  ; 出料手動允許信號
      AND     L168  ; 允許右IR輸送拉框昇降氣缸   伸出
      OUT     T168 D106  ; 手動右IR輸送拉框昇降氣缸上昇 / 出料爐體SW延遲時間
6829  LD      L3663  ; 出料自動允許信號
      AND     L4728  ; 右側合流拉框出料定點
      AND     L4731  ; 右側合流拉框夾爪開定點
      ANI     L4736  ; 右側合流拉框昇降上定點
      AND     L168  ; 允許右IR輸送拉框昇降氣缸   伸出
      OUT     T468 D107  ; 自動右IR輸送拉框昇降氣缸上昇 / 出料爐體自動延遲時間
6838  LD      B1168  ; 右IR輸送拉框昇降氣缸上昇
      AND     B253  ; 右IR輸送拉框下降氣缸C16縮回SV
      OR      T168  ; 手動右IR輸送拉框昇降氣缸上昇
      OR      T468  ; 自動右IR輸送拉框昇降氣缸上昇
      ANI     T169  ; 手動右IR輸送拉框昇降氣缸下降
      AND     L168  ; 允許右IR輸送拉框昇降氣缸   伸出
      ANI     L4736  ; 右側合流拉框昇降上定點
      OUT     B1168  ; 右IR輸送拉框昇降氣缸上昇
6846  LD      B1168  ; 右IR輸送拉框昇降氣缸上昇
      OUT     B253  ; 右IR輸送拉框下降氣缸C16縮回SV
6848  LD      B1168  ; 右IR輸送拉框昇降氣缸上昇
      AND     SM412  ; 1.0 Sec Clock
      OR      L4736  ; 右側合流拉框昇降上定點
      OUT     M368  ; 手動右IR輸送拉框昇降氣缸上昇燈
6852  LD      L4027  ; 出料機構允許運轉
      ANDPI   M4141  ; 右IR輸送拉框昇降異常
      OUT     L169  ; 允許右IR輸送拉框昇降氣缸縮回
6856  LD      M169  ; 右IR輸送拉框昇降下降SW
      AND     L3653  ; 出料手動允許信號
      AND     L169  ; 允許右IR輸送拉框昇降氣缸縮回
      OUT     T169 D106  ; 手動右IR輸送拉框昇降氣缸下降 / 出料爐體SW延遲時間
6863  LD      L3663  ; 出料自動允許信號
      AND     L4725  ; 右側合流補助昇降無框
      AND     L4727  ; 右側輸送出框定點無框
      AND     L4729  ; 右側合流拉框進料定點
      AND     L4731  ; 右側合流拉框夾爪開定點
      AND     L4751  ; 出料合流右側縮回定點
      ANI     L4735  ; 右側合流拉框昇降下定點
      AND     L169  ; 允許右IR輸送拉框昇降氣缸縮回
      ANI     M4143  ; 右側合流拉框掉框異常
      OUT     T469 D107  ; 自動右IR輸送拉框昇降氣缸下降 / 出料爐體自動延遲時間
